LIN {X -0.073,Y -233.852,Z 1712.235,A 0.000,B 0.000,C 90.000,E1 42.285} C_DIS
LIN {X -0.119,Y -224.509,Z 1712.218,A 0.000,B 0.000,C 90.000,E1 39.277} C_DIS
LIN {X 0.012,Y -216.138,Z 1712.201,A 0.000,B 0.000,C 90.000,E1 36.171} C_DIS
LIN {X 0.036,Y -208.461,Z 1712.184,A 0.000,B 0.000,C 90.000,E1 33.038} C_DIS
LIN {X -0.006,Y -201.606,Z 1712.166,A 0.000,B 0.000,C 90.000,E1 29.873} C_DIS
LIN {X 0.104,Y -195.298,Z 1712.148,A 0.000,B 0.000,C 90.000,E1 26.616} C_DIS
LIN {X -0.043,Y -188.244,Z 1712.125,A 0.000,B 0.000,C 90.000,E1 22.567} C_DIS
LIN {X 0.061,Y -183.297,Z 1712.107,A 0.000,B 0.000,C 90.000,E1 19.214} C_DIS
LIN {X -0.070,Y -179.154,Z 1712.088,A 0.000,B 0.000,C 90.000,E1 15.898} C_DIS
LIN {X -0.070,Y -174.908,Z 1712.065,A 0.000,B 0.000,C 90.000,E1 11.658} C_DIS
LIN {X 0.007,Y -171.641,Z 1712.041,A 0.000,B 0.000,C 90.000,E1 7.352} C_DIS
LIN {X -0.001,Y -169.062,Z 1712.012,A 0.000,B 0.000,C 90.000,E1 2.178} C_DIS
LIN {X 0.004,Y -167.943,Z 1711.964,A 0.000,B 0.000,C 90.000,E1 353.451} C_DIS
LIN {X -0.010,Y -169.850,Z 1711.920,A 0.000,B 0.000,C 90.000,E1 345.644} C_DIS
LIN {X -0.055,Y -172.730,Z 1711.891,A 0.000,B 0.000,C 90.000,E1 340.477} C_DIS
LIN {X -0.022,Y -176.262,Z 1711.868,A 0.000,B 0.000,C 90.000,E1 336.177} C_DIS
LIN {X 0.067,Y -180.723,Z 1711.844,A 0.000,B 0.000,C 90.000,E1 331.897} C_DIS
LIN {X 0.046,Y -185.271,Z 1711.825,A 0.000,B 0.000,C 90.000,E1 328.535} C_DIS
LIN {X -0.042,Y -190.788,Z 1711.807,A 0.000,B 0.000,C 90.000,E1 325.229} C_DIS
LIN {X -0.067,Y -195.689,Z 1711.793,A 0.000,B 0.000,C 90.000,E1 322.763} C_DIS
LIN {X -0.052,Y -202.307,Z 1711.777,A 0.000,B 0.000,C 90.000,E1 319.908} C_DIS
LIN {X 0.059,Y -208.732,Z 1711.764,A 0.000,B 0.000,C 90.000,E1 317.472} C_DIS
LIN {X -0.120,Y -217.156,Z 1711.748,A 0.000,B 0.000,C 90.000,E1 314.757} C_DIS
LIN {X -0.028,Y -225.299,Z 1711.736,A 0.000,B 0.000,C 90.000,E1 312.405} C_DIS
LIN {X 0.075,Y -234.395,Z 1711.723,A 0.000,B 0.000,C 90.000,E1 310.092} C_DIS
LIN {X -0.084,Y -242.909,Z 1711.712,A 0.000,B 0.000,C 90.000,E1 308.257} C_DIS
LIN {X 0.079,Y -250.460,Z 1711.704,A 0.000,B 0.000,C 90.000,E1 306.744} C_DIS
LIN {X -0.098,Y -262.879,Z 1711.692,A 0.000,B 0.000,C 90.000,E1 304.612} C_DIS
LIN {X -0.104,Y -281.105,Z 1711.677,A 0.000,B 0.000,C 90.000,E1 301.799} C_DIS
LIN {X -0.081,Y -300.693,Z 1711.661,A 0.000,B 0.000,C 90.000,E1 299.077} C_DIS
LIN {X 0.056,Y -315.955,Z 1711.651,A 0.000,B 0.000,C 90.000,E1 297.078} C_DIS
LIN {X 0.065,Y -331.490,Z 1711.640,A 0.000,B 0.000,C 90.000,E1 295.155} C_DIS
LIN {X 0.085,Y -344.408,Z 1711.631,A 0.000,B 0.000,C 90.000,E1 293.590} C_DIS
LIN {X 0.027,Y -359.701,Z 1711.621,A 0.000,B 0.000,C 90.000,E1 291.770} C_DIS
LIN {X -0.109,Y -371.942,Z 1711.613,A 0.000,B 0.000,C 90.000,E1 290.301} C_DIS
LIN {X 0.053,Y -378.776,Z 1711.608,A 0.000,B 0.000,C 90.000,E1 289.396} C_DIS
LIN {X -0.069,Y -384.788,Z 1711.603,A 0.000,B 0.000,C 90.000,E1 288.544} C_DIS
LIN {X 0.083,Y -388.314,Z 1711.600,A 0.000,B 0.000,C 90.000,E1 287.946} C_DIS
LIN {X -0.112,Y -391.399,Z 1711.597,A 0.000,B 0.000,C 90.000,E1 287.402} C_DIS
LIN {X 0.087,Y -394.052,Z 1711.593,A 0.000,B 0.000,C 90.000,E1 286.804} C_DIS
LIN {X -0.017,Y -397.255,Z 1711.589,A 0.000,B 0.000,C 90.000,E1 285.969} C_DIS
LIN {X -0.162,Y -398.955,Z 1711.586,A 0.000,B 0.000,C 90.000,E1 285.426} C_DIS
LIN {X 0.082,Y -400.312,Z 1711.582,A 0.000,B 0.000,C 90.000,E1 284.828} C_DIS
LIN {X -0.154,Y -401.245,Z 1711.579,A 0.000,B 0.000,C 90.000,E1 284.300} C_DIS
LIN {X 0.011,Y -401.838,Z 1711.576,A 0.000,B 0.000,C 90.000,E1 283.716} C_DIS
LIN {X -0.115,Y -402.031,Z 1711.573,A 0.000,B 0.000,C 90.000,E1 283.175} C_DIS
LIN {X 0.060,Y -401.772,Z 1711.570,A 0.000,B 0.000,C 90.000,E1 282.591} C_DIS
LIN {X -0.154,Y -401.091,Z 1711.567,A 0.000,B 0.000,C 90.000,E1 282.063} C_DIS
LIN {X 0.023,Y -399.884,Z 1711.564,A 0.000,B 0.000,C 90.000,E1 281.478} C_DIS
LIN {X 0.194,Y -398.188,Z 1711.561,A 0.000,B 0.000,C 90.000,E1 280.894} C_DIS
LIN {X -0.034,Y -395.932,Z 1711.558,A 0.000,B 0.000,C 90.000,E1 280.366} C_DIS
LIN {X 0.044,Y -393.111,Z 1711.554,A 0.000,B 0.000,C 90.000,E1 279.792} C_DIS
LIN {X -0.158,Y -388.091,Z 1711.550,A 0.000,B 0.000,C 90.000,E1 278.973} C_DIS
LIN {X -0.066,Y -379.299,Z 1711.542,A 0.000,B 0.000,C 90.000,E1 277.530} C_DIS
LIN {X -0.066,Y -373.299,Z 1711.537,A 0.000,B 0.000,C 90.000,E1 276.663} C_DIS
LIN {X -0.107,Y -368.624,Z 1711.534,A 0.000,B 0.000,C 90.000,E1 276.087} C_DIS
LIN {X -0.152,Y -363.231,Z 1711.531,A 0.000,B 0.000,C 90.000,E1 275.511} C_DIS
LIN {X -0.040,Y -357.396,Z 1711.527,A 0.000,B 0.000,C 90.000,E1 274.935} C_DIS
LIN {X -0.006,Y -351.283,Z 1711.525,A 0.000,B 0.000,C 90.000,E1 274.416} C_DIS
LIN {X -0.054,Y -345.014,Z 1711.522,A 0.000,B 0.000,C 90.000,E1 273.955} C_DIS
LIN {X 0.142,Y -338.578,Z 1711.520,A 0.000,B 0.000,C 90.000,E1 273.498} C_DIS
LIN {X -0.083,Y -332.051,Z 1711.517,A 0.000,B 0.000,C 90.000,E1 273.154} C_DIS
LIN {X -0.060,Y -325.544,Z 1711.516,A 0.000,B 0.000,C 90.000,E1 272.808} C_DIS
LIN {X 0.149,Y -318.882,Z 1711.514,A 0.000,B 0.000,C 90.000,E1 272.465} C_DIS
LIN {X -0.098,Y -312.037,Z 1711.512,A 0.000,B 0.000,C 90.000,E1 272.236} C_DIS
LIN {X -0.141,Y -301.639,Z 1711.510,A 0.000,B 0.000,C 90.000,E1 271.892} C_DIS
LIN {X 0.131,Y -290.878,Z 1711.509,A 0.000,B 0.000,C 90.000,E1 271.547} C_DIS
LIN {X 0.080,Y -279.215,Z 1711.507,A 0.000,B 0.000,C 90.000,E1 271.318} C_DIS
LIN {X -0.015,Y -266.610,Z 1711.506,A 0.000,B 0.000,C 90.000,E1 271.146} C_DIS
LIN {X 0.035,Y -256.490,Z 1711.506,A 0.000,B 0.000,C 90.000,E1 271.031} C_DIS
LIN {X 0.100,Y -247.221,Z 1711.505,A 0.000,B 0.000,C 90.000,E1 270.974} C_DIS
LIN {X 0.052,Y -181.458,Z 1711.505,A 0.000,B 0.000,C 90.000,E1 270.974} C_DIS
LIN {X -0.077,Y -181.557,Z 1711.500,A 0.000,B 0.000,C 90.000,E1 270.000} C_DIS
LIN {X -0.075,Y -180.789,Z 1711.471,A 0.000,B 0.000,C 90.000,E1 264.780} C_DIS
LIN {X 0.000,Y -178.887,Z 1711.443,A 0.000,B 0.000,C 90.000,E1 259.690} C_DIS
LIN {X 0.075,Y -175.930,Z 1711.414,A 0.000,B 0.000,C 90.000,E1 254.574} C_DIS
LIN {X 0.020,Y -175.373,Z 1711.410,A 0.000,B 0.000,C 90.000,E1 253.740} C_DIS
LIN {X 0.079,Y -172.149,Z 1711.386,A 0.000,B 0.000,C 90.000,E1 249.444} C_DIS
LIN {X 0.056,Y -171.615,Z 1711.381,A 0.000,B 0.000,C 90.000,E1 248.592} C_DIS
LIN {X 0.044,Y -167.837,Z 1711.357,A 0.000,B 0.000,C 90.000,E1 244.280} C_DIS
LIN {X 0.061,Y -166.564,Z 1711.348,A 0.000,B 0.000,C 90.000,E1 242.538} C_DIS
LIN {X -0.029,Y -162.558,Z 1711.323,A 0.000,B 0.000,C 90.000,E1 238.201} C_DIS
LIN {X 0.031,Y -161.237,Z 1711.313,A 0.000,B 0.000,C 90.000,E1 236.421} C_DIS
LIN {X 0.065,Y -157.242,Z 1711.289,A 0.000,B 0.000,C 90.000,E1 231.984} C_DIS
LIN {X -0.012,Y -155.965,Z 1711.279,A 0.000,B 0.000,C 90.000,E1 230.231} C_DIS
LIN {X 0.046,Y -152.220,Z 1711.254,A 0.000,B 0.000,C 90.000,E1 225.729} C_DIS
LIN {X 0.067,Y -150.463,Z 1711.239,A 0.000,B 0.000,C 90.000,E1 223.014} C_DIS
LIN {X -0.022,Y -147.188,Z 1711.214,A 0.000,B 0.000,C 90.000,E1 218.508} C_DIS
LIN {X 0.059,Y -145.207,Z 1711.194,A 0.000,B 0.000,C 90.000,E1 214.818} C_DIS
LIN {X -0.031,Y -142.341,Z 1711.163,A 0.000,B 0.000,C 90.000,E1 209.333} C_DIS
LIN {X 0.022,Y -141.730,Z 1711.153,A 0.000,B 0.000,C 90.000,E1 207.462} C_DIS
LIN {X 0.004,Y -139.482,Z 1711.117,A 0.000,B 0.000,C 90.000,E1 200.972} C_DIS
LIN {X -0.007,Y -138.982,Z 1711.101,A 0.000,B 0.000,C 90.000,E1 198.181} C_DIS
LIN {X -0.045,Y -138.333,Z 1711.054,A 0.000,B 0.000,C 90.000,E1 189.792} C_DIS
LIN {X -0.022,Y -139.428,Z 1711.008,A 0.000,B 0.000,C 90.000,E1 181.375} C_DIS
LIN {X 0.032,Y -141.353,Z 1710.971,A 0.000,B 0.000,C 90.000,E1 174.837} C_DIS
LIN {X 0.008,Y -142.706,Z 1710.956,A 0.000,B 0.000,C 90.000,E1 172.064} C_DIS
LIN {X -0.033,Y -145.079,Z 1710.930,A 0.000,B 0.000,C 90.000,E1 167.465} C_DIS
LIN {X -0.038,Y -147.704,Z 1710.910,A 0.000,B 0.000,C 90.000,E1 163.795} C_DIS
LIN {X 0.047,Y -150.357,Z 1710.890,A 0.000,B 0.000,C 90.000,E1 160.115} C_DIS
LIN {X 0.066,Y -153.782,Z 1710.870,A 0.000,B 0.000,C 90.000,E1 156.485} C_DIS
LIN {X -0.015,Y -157.194,Z 1710.849,A 0.000,B 0.000,C 90.000,E1 152.922} C_DIS
LIN {X 0.068,Y -161.354,Z 1710.830,A 0.000,B 0.000,C 90.000,E1 149.331} C_DIS
LIN {X 0.079,Y -165.557,Z 1710.810,A 0.000,B 0.000,C 90.000,E1 145.801} C_DIS
LIN {X -0.037,Y -170.473,Z 1710.791,A 0.000,B 0.000,C 90.000,E1 142.351} C_DIS
LIN {X 0.113,Y -175.355,Z 1710.772,A 0.000,B 0.000,C 90.000,E1 138.852} C_DIS
LIN {X -0.024,Y -180.979,Z 1710.753,A 0.000,B 0.000,C 90.000,E1 135.486} C_DIS
LIN {X -0.037,Y -186.404,Z 1710.734,A 0.000,B 0.000,C 90.000,E1 132.123} C_DIS
LIN {X -0.098,Y -191.032,Z 1710.720,A 0.000,B 0.000,C 90.000,E1 129.644} C_DIS
LIN {X 0.094,Y -196.814,Z 1710.702,A 0.000,B 0.000,C 90.000,E1 126.297} C_DIS
LIN {X 0.013,Y -200.068,Z 1710.693,A 0.000,B 0.000,C 90.000,E1 124.692} C_DIS
LIN {X 0.007,Y -207.567,Z 1710.670,A 0.000,B 0.000,C 90.000,E1 120.669} C_DIS
LIN {X -0.063,Y -209.260,Z 1710.666,A 0.000,B 0.000,C 90.000,E1 119.873} C_DIS
LIN {X -0.135,Y -332.673,Z 1710.666,A 0.000,B 0.000,C 90.000,E1 119.873} C_DIS
LIN {X 0.115,Y -334.980,Z 1710.666,A 0.000,B 0.000,C 90.000,E1 119.795} C_DIS
LIN {X 0.082,Y -339.177,Z 1710.665,A 0.000,B 0.000,C 90.000,E1 119.617} C_DIS
LIN {X -0.082,Y -341.592,Z 1710.664,A 0.000,B 0.000,C 90.000,E1 119.461} C_DIS
LIN {X 0.017,Y -344.886,Z 1710.661,A 0.000,B 0.000,C 90.000,E1 119.077} C_DIS
LIN {X 0.075,Y -346.788,Z 1710.660,A 0.000,B 0.000,C 90.000,E1 118.771} C_DIS
LIN {X -0.129,Y -350.995,Z 1710.655,A 0.000,B 0.000,C 90.000,E1 117.897} C_DIS
LIN {X 0.064,Y -364.150,Z 1710.640,A 0.000,B 0.000,C 90.000,E1 115.155} C_DIS
LIN {X -0.005,Y -378.851,Z 1710.625,A 0.000,B 0.000,C 90.000,E1 112.514} C_DIS
LIN {X 0.106,Y -393.315,Z 1710.612,A 0.000,B 0.000,C 90.000,E1 110.194} C_DIS
LIN {X 0.084,Y -409.198,Z 1710.600,A 0.000,B 0.000,C 90.000,E1 107.946} C_DIS
LIN {X -0.207,Y -426.609,Z 1710.588,A 0.000,B 0.000,C 90.000,E1 105.788} C_DIS
LIN {X -0.198,Y -445.654,Z 1710.576,A 0.000,B 0.000,C 90.000,E1 103.647} C_DIS
LIN {X 0.226,Y -465.672,Z 1710.565,A 0.000,B 0.000,C 90.000,E1 101.591} C_DIS
LIN {X 0.014,Y -488.822,Z 1710.553,A 0.000,B 0.000,C 90.000,E1 99.557} C_DIS
LIN {X 0.092,Y -504.598,Z 1710.546,A 0.000,B 0.000,C 90.000,E1 98.276} C_DIS
LIN {X -0.221,Y -507.002,Z 1710.545,A 0.000,B 0.000,C 90.000,E1 98.106} C_DIS
LIN {X 0.003,Y -510.391,Z 1710.542,A 0.000,B 0.000,C 90.000,E1 97.644} C_DIS
LIN {X -0.052,Y -511.618,Z 1710.541,A 0.000,B 0.000,C 90.000,E1 97.409} C_DIS
LIN {X -0.173,Y -512.507,Z 1710.540,A 0.000,B 0.000,C 90.000,E1 97.182} C_DIS
LIN {X 0.186,Y -513.424,Z 1710.537,A 0.000,B 0.000,C 90.000,E1 96.663} C_DIS
LIN {X 0.040,Y -513.316,Z 1710.534,A 0.000,B 0.000,C 90.000,E1 96.201} C_DIS
LIN {X -0.102,Y -512.160,Z 1710.532,A 0.000,B 0.000,C 90.000,E1 95.739} C_DIS
LIN {X -0.197,Y -511.132,Z 1710.531,A 0.000,B 0.000,C 90.000,E1 95.511} C_DIS
LIN {X -0.244,Y -509.734,Z 1710.529,A 0.000,B 0.000,C 90.000,E1 95.277} C_DIS
LIN {X 0.075,Y -497.149,Z 1710.520,A 0.000,B 0.000,C 90.000,E1 93.555} C_DIS
LIN {X 0.125,Y -484.524,Z 1710.510,A 0.000,B 0.000,C 90.000,E1 91.835} C_DIS
LIN {X -0.077,Y -471.809,Z 1710.501,A 0.000,B 0.000,C 90.000,E1 90.115} C_DIS
LIN {X -0.063,Y -458.968,Z 1710.491,A 0.000,B 0.000,C 90.000,E1 88.339} C_DIS
LIN {X 0.168,Y -445.987,Z 1710.481,A 0.000,B 0.000,C 90.000,E1 86.502} C_DIS
LIN {X 0.139,Y -433.000,Z 1710.470,A 0.000,B 0.000,C 90.000,E1 84.666} C_DIS
LIN {X 0.168,Y -416.433,Z 1710.457,A 0.000,B 0.000,C 90.000,E1 82.243} C_DIS
LIN {X 0.081,Y -397.068,Z 1710.440,A 0.000,B 0.000,C 90.000,E1 79.218} C_DIS
LIN {X -0.139,Y -382.139,Z 1710.426,A 0.000,B 0.000,C 90.000,E1 76.700} C_DIS
LIN {X -0.205,Y -367.739,Z 1710.411,A 0.000,B 0.000,C 90.000,E1 74.102} C_DIS
LIN {X 0.047,Y -355.320,Z 1710.398,A 0.000,B 0.000,C 90.000,E1 71.692} C_DIS
LIN {X 0.136,Y -340.409,Z 1710.381,A 0.000,B 0.000,C 90.000,E1 68.646} C_DIS
LIN {X 0.072,Y -328.886,Z 1710.368,A 0.000,B 0.000,C 90.000,E1 66.177} C_DIS
LIN {X 0.050,Y -316.355,Z 1710.352,A 0.000,B 0.000,C 90.000,E1 63.332} C_DIS
LIN {X -0.197,Y -305.422,Z 1710.338,A 0.000,B 0.000,C 90.000,E1 60.795} C_DIS
LIN {X 0.010,Y -294.627,Z 1710.323,A 0.000,B 0.000,C 90.000,E1 58.122} C_DIS
LIN {X 0.135,Y -286.448,Z 1710.312,A 0.000,B 0.000,C 90.000,E1 56.087} C_DIS
LIN {X 0.022,Y -278.092,Z 1710.300,A 0.000,B 0.000,C 90.000,E1 54.069} C_DIS
LIN {X -0.041,Y -268.222,Z 1710.287,A 0.000,B 0.000,C 90.000,E1 51.662} C_DIS
LIN {X 0.050,Y -258.392,Z 1710.273,A 0.000,B 0.000,C 90.000,E1 49.175} C_DIS
LIN {X 0.053,Y -247.517,Z 1710.257,A 0.000,B 0.000,C 90.000,E1 46.296} C_DIS
LIN {X -0.064,Y -235.971,Z 1710.239,A 0.000,B 0.000,C 90.000,E1 43.014} C_DIS
LIN {X -0.134,Y -225.354,Z 1710.220,A 0.000,B 0.000,C 90.000,E1 39.644} C_DIS
LIN {X -0.060,Y -215.903,Z 1710.201,A 0.000,B 0.000,C 90.000,E1 36.171} C_DIS
LIN {X -0.039,Y -208.266,Z 1710.183,A 0.000,B 0.000,C 90.000,E1 33.038} C_DIS
LIN {X -0.082,Y -201.421,Z 1710.166,A 0.000,B 0.000,C 90.000,E1 29.873} C_DIS
LIN {X 0.026,Y -195.152,Z 1710.148,A 0.000,B 0.000,C 90.000,E1 26.616} C_DIS
LIN {X 0.051,Y -188.122,Z 1710.125,A 0.000,B 0.000,C 90.000,E1 22.514} C_DIS
LIN {X -0.020,Y -183.190,Z 1710.107,A 0.000,B 0.000,C 90.000,E1 19.214} C_DIS
LIN {X 0.021,Y -179.067,Z 1710.088,A 0.000,B 0.000,C 90.000,E1 15.843} C_DIS
LIN {X 0.055,Y -174.829,Z 1710.064,A 0.000,B 0.000,C 90.000,E1 11.591} C_DIS
LIN {X -0.076,Y -171.580,Z 1710.041,A 0.000,B 0.000,C 90.000,E1 7.352} C_DIS
LIN {X -0.085,Y -169.011,Z 1710.012,A 0.000,B 0.000,C 90.000,E1 2.178} C_DIS
LIN {X 0.002,Y -167.882,Z 1709.964,A 0.000,B 0.000,C 90.000,E1 353.451} C_DIS
LIN {X -0.017,Y -169.793,Z 1709.920,A 0.000,B 0.000,C 90.000,E1 345.644} C_DIS
LIN {X 0.099,Y -172.653,Z 1709.891,A 0.000,B 0.000,C 90.000,E1 340.423} C_DIS
LIN {X -0.032,Y -176.218,Z 1709.868,A 0.000,B 0.000,C 90.000,E1 336.177} C_DIS
LIN {X 0.055,Y -180.714,Z 1709.844,A 0.000,B 0.000,C 90.000,E1 331.897} C_DIS
LIN {X 0.033,Y -185.287,Z 1709.825,A 0.000,B 0.000,C 90.000,E1 328.535} C_DIS
LIN {X 0.102,Y -190.854,Z 1709.807,A 0.000,B 0.000,C 90.000,E1 325.182} C_DIS
LIN {X -0.079,Y -195.788,Z 1709.793,A 0.000,B 0.000,C 90.000,E1 322.763} C_DIS
LIN {X -0.062,Y -202.412,Z 1709.777,A 0.000,B 0.000,C 90.000,E1 319.908} C_DIS
LIN {X 0.050,Y -208.879,Z 1709.764,A 0.000,B 0.000,C 90.000,E1 317.472} C_DIS
LIN {X 0.027,Y -217.335,Z 1709.748,A 0.000,B 0.000,C 90.000,E1 314.717} C_DIS
LIN {X -0.031,Y -225.515,Z 1709.736,A 0.000,B 0.000,C 90.000,E1 312.405} C_DIS
LIN {X 0.077,Y -234.626,Z 1709.723,A 0.000,B 0.000,C 90.000,E1 310.092} C_DIS
LIN {X -0.078,Y -243.148,Z 1709.712,A 0.000,B 0.000,C 90.000,E1 308.257} C_DIS
LIN {X -0.113,Y -250.680,Z 1709.704,A 0.000,B 0.000,C 90.000,E1 306.790} C_DIS
LIN {X -0.084,Y -263.090,Z 1709.692,A 0.000,B 0.000,C 90.000,E1 304.612} C_DIS
LIN {X -0.085,Y -281.271,Z 1709.677,A 0.000,B 0.000,C 90.000,E1 301.799} C_DIS
LIN {X -0.055,Y -300.825,Z 1709.661,A 0.000,B 0.000,C 90.000,E1 299.077} C_DIS
LIN {X 0.085,Y -316.083,Z 1709.651,A 0.000,B 0.000,C 90.000,E1 297.078} C_DIS
LIN {X 0.099,Y -331.545,Z 1709.640,A 0.000,B 0.000,C 90.000,E1 295.155} C_DIS
LIN {X -0.196,Y -344.452,Z 1709.631,A 0.000,B 0.000,C 90.000,E1 293.643} C_DIS
LIN {X 0.100,Y -359.701,Z 1709.621,A 0.000,B 0.000,C 90.000,E1 291.770} C_DIS
LIN {X -0.123,Y -369.594,Z 1709.614,A 0.000,B 0.000,C 90.000,E1 290.610} C_DIS
LIN {X 0.023,Y -376.566,Z 1709.609,A 0.000,B 0.000,C 90.000,E1 289.704} C_DIS
LIN {X -0.116,Y -380.869,Z 1709.606,A 0.000,B 0.000,C 90.000,E1 289.141} C_DIS
LIN {X 0.007,Y -384.821,Z 1709.603,A 0.000,B 0.000,C 90.000,E1 288.544} C_DIS
LIN {X -0.211,Y -388.386,Z 1709.600,A 0.000,B 0.000,C 90.000,E1 288.000} C_DIS
LIN {X -0.035,Y -391.476,Z 1709.597,A 0.000,B 0.000,C 90.000,E1 287.402} C_DIS
LIN {X 0.164,Y -394.104,Z 1709.594,A 0.000,B 0.000,C 90.000,E1 286.804} C_DIS
LIN {X 0.060,Y -397.394,Z 1709.589,A 0.000,B 0.000,C 90.000,E1 285.969} C_DIS
LIN {X -0.082,Y -399.087,Z 1709.586,A 0.000,B 0.000,C 90.000,E1 285.426} C_DIS
LIN {X 0.163,Y -400.457,Z 1709.583,A 0.000,B 0.000,C 90.000,E1 284.828} C_DIS
LIN {X -0.072,Y -401.431,Z 1709.579,A 0.000,B 0.000,C 90.000,E1 284.300} C_DIS
LIN {X 0.094,Y -402.004,Z 1709.576,A 0.000,B 0.000,C 90.000,E1 283.716} C_DIS
LIN {X -0.031,Y -402.214,Z 1709.573,A 0.000,B 0.000,C 90.000,E1 283.175} C_DIS
LIN {X 0.145,Y -401.980,Z 1709.570,A 0.000,B 0.000,C 90.000,E1 282.591} C_DIS
LIN {X -0.068,Y -401.298,Z 1709.567,A 0.000,B 0.000,C 90.000,E1 282.063} C_DIS
LIN {X 0.110,Y -400.154,Z 1709.564,A 0.000,B 0.000,C 90.000,E1 281.478} C_DIS
LIN {X -0.109,Y -398.447,Z 1709.561,A 0.000,B 0.000,C 90.000,E1 280.950} C_DIS
LIN {X 0.055,Y -396.218,Z 1709.558,A 0.000,B 0.000,C 90.000,E1 280.366} C_DIS
LIN {X 0.134,Y -393.406,Z 1709.555,A 0.000,B 0.000,C 90.000,E1 279.792} C_DIS
LIN {X -0.066,Y -388.456,Z 1709.550,A 0.000,B 0.000,C 90.000,E1 278.973} C_DIS
LIN {X 0.029,Y -379.616,Z 1709.542,A 0.000,B 0.000,C 90.000,E1 277.530} C_DIS
LIN {X 0.030,Y -373.544,Z 1709.537,A 0.000,B 0.000,C 90.000,E1 276.663} C_DIS
LIN {X -0.011,Y -368.837,Z 1709.534,A 0.000,B 0.000,C 90.000,E1 276.087} C_DIS
LIN {X -0.062,Y -363.443,Z 1709.531,A 0.000,B 0.000,C 90.000,E1 275.511} C_DIS
LIN {X 0.058,Y -357.562,Z 1709.527,A 0.000,B 0.000,C 90.000,E1 274.935} C_DIS
LIN {X 0.116,Y -351.452,Z 1709.525,A 0.000,B 0.000,C 90.000,E1 274.416} C_DIS
LIN {X 0.084,Y -345.215,Z 1709.522,A 0.000,B 0.000,C 90.000,E1 273.955} C_DIS
LIN {X -0.049,Y -338.811,Z 1709.520,A 0.000,B 0.000,C 90.000,E1 273.555} C_DIS
LIN {X 0.075,Y -332.277,Z 1709.518,A 0.000,B 0.000,C 90.000,E1 273.154} C_DIS
LIN {X 0.096,Y -325.680,Z 1709.516,A 0.000,B 0.000,C 90.000,E1 272.808} C_DIS
LIN {X -0.034,Y -318.935,Z 1709.514,A 0.000,B 0.000,C 90.000,E1 272.522} C_DIS
LIN {X 0.041,Y -312.097,Z 1709.512,A 0.000,B 0.000,C 90.000,E1 272.236} C_DIS
LIN {X 0.020,Y -301.843,Z 1709.510,A 0.000,B 0.000,C 90.000,E1 271.892} C_DIS
LIN {X -0.010,Y -291.070,Z 1709.509,A 0.000,B 0.000,C 90.000,E1 271.604} C_DIS
LIN {X -0.052,Y -279.680,Z 1709.508,A 0.000,B 0.000,C 90.000,E1 271.375} C_DIS
LIN {X 0.113,Y -267.186,Z 1709.506,A 0.000,B 0.000,C 90.000,E1 271.146} C_DIS
LIN {X -0.102,Y -256.616,Z 1709.506,A 0.000,B 0.000,C 90.000,E1 271.088} C_DIS
LIN {X -0.031,Y -247.213,Z 1709.506,A 0.000,B 0.000,C 90.000,E1 271.031} C_DIS
LIN {X -0.045,Y -181.452,Z 1709.506,A 0.000,B 0.000,C 90.000,E1 271.031} C_DIS
LIN {X 0.008,Y -181.561,Z 1709.500,A 0.000,B 0.000,C 90.000,E1 270.000} C_DIS
LIN {X 0.010,Y -180.799,Z 1709.471,A 0.000,B 0.000,C 90.000,E1 264.780} C_DIS
LIN {X 0.083,Y -178.899,Z 1709.443,A 0.000,B 0.000,C 90.000,E1 259.690} C_DIS
LIN {X -0.012,Y -175.941,Z 1709.415,A 0.000,B 0.000,C 90.000,E1 254.629} C_DIS
LIN {X -0.065,Y -175.398,Z 1709.410,A 0.000,B 0.000,C 90.000,E1 253.795} C_DIS
LIN {X -0.061,Y -172.166,Z 1709.386,A 0.000,B 0.000,C 90.000,E1 249.518} C_DIS
LIN {X -0.022,Y -171.635,Z 1709.381,A 0.000,B 0.000,C 90.000,E1 248.646} C_DIS
LIN {X -0.026,Y -167.858,Z 1709.357,A 0.000,B 0.000,C 90.000,E1 244.332} C_DIS
LIN {X -0.083,Y -166.590,Z 1709.348,A 0.000,B 0.000,C 90.000,E1 242.615} C_DIS
LIN {X 0.051,Y -162.580,Z 1709.323,A 0.000,B 0.000,C 90.000,E1 238.201} C_DIS
LIN {X 0.020,Y -161.262,Z 1709.314,A 0.000,B 0.000,C 90.000,E1 236.453} C_DIS
LIN {X 0.019,Y -157.263,Z 1709.289,A 0.000,B 0.000,C 90.000,E1 232.029} C_DIS
LIN {X -0.055,Y -155.984,Z 1709.279,A 0.000,B 0.000,C 90.000,E1 230.275} C_DIS
LIN {X -0.093,Y -152.241,Z 1709.254,A 0.000,B 0.000,C 90.000,E1 225.810} C_DIS
LIN {X 0.033,Y -150.481,Z 1709.239,A 0.000,B 0.000,C 90.000,E1 223.056} C_DIS
LIN {X -0.040,Y -147.206,Z 1709.214,A 0.000,B 0.000,C 90.000,E1 218.543} C_DIS
LIN {X -0.069,Y -145.226,Z 1709.194,A 0.000,B 0.000,C 90.000,E1 214.898} C_DIS
LIN {X 0.041,Y -142.352,Z 1709.163,A 0.000,B 0.000,C 90.000,E1 209.333} C_DIS
LIN {X -0.031,Y -141.740,Z 1709.153,A 0.000,B 0.000,C 90.000,E1 207.513} C_DIS
LIN {X 0.076,Y -139.487,Z 1709.117,A 0.000,B 0.000,C 90.000,E1 200.972} C_DIS
LIN {X 0.064,Y -138.989,Z 1709.101,A 0.000,B 0.000,C 90.000,E1 198.181} C_DIS
LIN {X 0.026,Y -138.335,Z 1709.054,A 0.000,B 0.000,C 90.000,E1 189.792} C_DIS
LIN {X 0.050,Y -139.420,Z 1709.008,A 0.000,B 0.000,C 90.000,E1 181.375} C_DIS
LIN {X -0.037,Y -141.339,Z 1708.972,A 0.000,B 0.000,C 90.000,E1 174.894} C_DIS
LIN {X -0.079,Y -142.695,Z 1708.956,A 0.000,B 0.000,C 90.000,E1 172.129} C_DIS
LIN {X 0.041,Y -145.061,Z 1708.930,A 0.000,B 0.000,C 90.000,E1 167.465} C_DIS
LIN {X 0.038,Y -147.686,Z 1708.910,A 0.000,B 0.000,C 90.000,E1 163.795} C_DIS
LIN {X -0.070,Y -150.334,Z 1708.890,A 0.000,B 0.000,C 90.000,E1 160.188} C_DIS
LIN {X 0.001,Y -153.751,Z 1708.870,A 0.000,B 0.000,C 90.000,E1 156.538} C_DIS
LIN {X -0.008,Y -157.164,Z 1708.850,A 0.000,B 0.000,C 90.000,E1 152.948} C_DIS
LIN {X -0.074,Y -161.318,Z 1708.830,A 0.000,B 0.000,C 90.000,E1 149.410} C_DIS
LIN {X 0.080,Y -164.432,Z 1708.815,A 0.000,B 0.000,C 90.000,E1 146.707} C_DIS
LIN {X 0.073,Y -169.119,Z 1708.796,A 0.000,B 0.000,C 90.000,E1 143.210} C_DIS
LIN {X 0.022,Y -171.672,Z 1708.786,A 0.000,B 0.000,C 90.000,E1 141.492} C_DIS
LIN {X -0.067,Y -176.640,Z 1708.767,A 0.000,B 0.000,C 90.000,E1 138.081} C_DIS
LIN {X 0.061,Y -180.937,Z 1708.753,A 0.000,B 0.000,C 90.000,E1 135.486} C_DIS
LIN {X 0.050,Y -186.357,Z 1708.734,A 0.000,B 0.000,C 90.000,E1 132.123} C_DIS
LIN {X -0.010,Y -190.988,Z 1708.720,A 0.000,B 0.000,C 90.000,E1 129.644} C_DIS
LIN {X -0.092,Y -196.764,Z 1708.702,A 0.000,B 0.000,C 90.000,E1 126.377} C_DIS
LIN {X -0.061,Y -200.013,Z 1708.693,A 0.000,B 0.000,C 90.000,E1 124.739} C_DIS
LIN {X 0.099,Y -207.516,Z 1708.671,A 0.000,B 0.000,C 90.000,E1 120.669} C_DIS
LIN {X 0.074,Y -209.181,Z 1708.666,A 0.000,B 0.000,C 90.000,E1 119.873} C_DIS
LIN {X 0.083,Y -332.295,Z 1708.666,A 0.000,B 0.000,C 90.000,E1 119.873} C_DIS
LIN {X -0.194,Y -335.216,Z 1708.666,A 0.000,B 0.000,C 90.000,E1 119.873} C_DIS
LIN {X -0.063,Y -339.167,Z 1708.665,A 0.000,B 0.000,C 90.000,E1 119.667} C_DIS
LIN {X 0.069,Y -341.531,Z 1708.664,A 0.000,B 0.000,C 90.000,E1 119.461} C_DIS
LIN {X 0.168,Y -344.782,Z 1708.662,A 0.000,B 0.000,C 90.000,E1 119.077} C_DIS
LIN {X -0.093,Y -346.682,Z 1708.660,A 0.000,B 0.000,C 90.000,E1 118.821} C_DIS
LIN {X 0.011,Y -352.269,Z 1708.653,A 0.000,B 0.000,C 90.000,E1 117.590} C_DIS
LIN {X -0.079,Y -365.583,Z 1708.638,A 0.000,B 0.000,C 90.000,E1 114.899} C_DIS
LIN {X -0.112,Y -380.447,Z 1708.624,A 0.000,B 0.000,C 90.000,E1 112.259} C_DIS
LIN {X 0.029,Y -395.071,Z 1708.611,A 0.000,B 0.000,C 90.000,E1 109.939} C_DIS
LIN {X 0.039,Y -411.126,Z 1708.598,A 0.000,B 0.000,C 90.000,E1 107.692} C_DIS
LIN {X 0.194,Y -428.723,Z 1708.586,A 0.000,B 0.000,C 90.000,E1 105.481} C_DIS
LIN {X 0.191,Y -447.928,Z 1708.574,A 0.000,B 0.000,C 90.000,E1 103.355} C_DIS
LIN {X -0.216,Y -468.013,Z 1708.563,A 0.000,B 0.000,C 90.000,E1 101.422} C_DIS
LIN {X -0.211,Y -491.255,Z 1708.552,A 0.000,B 0.000,C 90.000,E1 99.378} C_DIS
LIN {X 0.203,Y -504.404,Z 1708.546,A 0.000,B 0.000,C 90.000,E1 98.276} C_DIS
LIN {X -0.111,Y -506.800,Z 1708.545,A 0.000,B 0.000,C 90.000,E1 98.106} C_DIS
LIN {X 0.031,Y -508.717,Z 1708.544,A 0.000,B 0.000,C 90.000,E1 97.871} C_DIS
LIN {X 0.104,Y -510.183,Z 1708.542,A 0.000,B 0.000,C 90.000,E1 97.644} C_DIS
LIN {X 0.054,Y -511.402,Z 1708.541,A 0.000,B 0.000,C 90.000,E1 97.409} C_DIS
LIN {X -0.063,Y -512.284,Z 1708.540,A 0.000,B 0.000,C 90.000,E1 97.182} C_DIS
LIN {X -0.215,Y -513.195,Z 1708.537,A 0.000,B 0.000,C 90.000,E1 96.720} C_DIS
LIN {X 0.148,Y -513.081,Z 1708.535,A 0.000,B 0.000,C 90.000,E1 96.201} C_DIS
LIN {X 0.005,Y -511.920,Z 1708.532,A 0.000,B 0.000,C 90.000,E1 95.739} C_DIS
LIN {X -0.091,Y -510.890,Z 1708.531,A 0.000,B 0.000,C 90.000,E1 95.511} C_DIS
LIN {X -0.139,Y -509.488,Z 1708.529,A 0.000,B 0.000,C 90.000,E1 95.277} C_DIS
LIN {X 0.172,Y -496.899,Z 1708.520,A 0.000,B 0.000,C 90.000,E1 93.555} C_DIS
LIN {X 0.214,Y -484.285,Z 1708.510,A 0.000,B 0.000,C 90.000,E1 91.835} C_DIS
LIN {X 0.007,Y -471.582,Z 1708.501,A 0.000,B 0.000,C 90.000,E1 90.115} C_DIS
LIN {X 0.013,Y -458.748,Z 1708.491,A 0.000,B 0.000,C 90.000,E1 88.339} C_DIS
LIN {X -0.207,Y -445.766,Z 1708.481,A 0.000,B 0.000,C 90.000,E1 86.560} C_DIS
LIN {X 0.202,Y -432.745,Z 1708.470,A 0.000,B 0.000,C 90.000,E1 84.666} C_DIS
LIN {X -0.189,Y -416.155,Z 1708.457,A 0.000,B 0.000,C 90.000,E1 82.299} C_DIS
LIN {X 0.124,Y -396.765,Z 1708.440,A 0.000,B 0.000,C 90.000,E1 79.218} C_DIS
LIN {X -0.106,Y -381.820,Z 1708.426,A 0.000,B 0.000,C 90.000,E1 76.700} C_DIS
LIN {X -0.181,Y -367.393,Z 1708.411,A 0.000,B 0.000,C 90.000,E1 74.102} C_DIS
LIN {X 0.061,Y -354.939,Z 1708.398,A 0.000,B 0.000,C 90.000,E1 71.692} C_DIS
LIN {X 0.139,Y -340.019,Z 1708.381,A 0.000,B 0.000,C 90.000,E1 68.646} C_DIS
LIN {X 0.087,Y -329.937,Z 1708.370,A 0.000,B 0.000,C 90.000,E1 66.485} C_DIS
LIN {X 0.103,Y -317.363,Z 1708.354,A 0.000,B 0.000,C 90.000,E1 63.640} C_DIS
LIN {X 0.153,Y -306.425,Z 1708.339,A 0.000,B 0.000,C 90.000,E1 61.051} C_DIS
LIN {X -0.047,Y -296.966,Z 1708.327,A 0.000,B 0.000,C 90.000,E1 58.791} C_DIS
LIN {X -0.031,Y -288.862,Z 1708.315,A 0.000,B 0.000,C 90.000,E1 56.786} C_DIS
LIN {X -0.095,Y -280.542,Z 1708.304,A 0.000,B 0.000,C 90.000,E1 54.769} C_DIS
LIN {X 0.016,Y -272.100,Z 1708.293,A 0.000,B 0.000,C 90.000,E1 52.683} C_DIS
LIN {X 0.032,Y -262.245,Z 1708.279,A 0.000,B 0.000,C 90.000,E1 50.231} C_DIS
LIN {X -0.022,Y -249.840,Z 1708.261,A 0.000,B 0.000,C 90.000,E1 47.025} C_DIS
LIN {X 0.088,Y -238.126,Z 1708.243,A 0.000,B 0.000,C 90.000,E1 43.704} C_DIS
LIN {X 0.068,Y -227.351,Z 1708.224,A 0.000,B 0.000,C 90.000,E1 40.334} C_DIS
LIN {X -0.021,Y -219.737,Z 1708.209,A 0.000,B 0.000,C 90.000,E1 37.684} C_DIS
LIN {X -0.131,Y -211.754,Z 1708.192,A 0.000,B 0.000,C 90.000,E1 34.612} C_DIS
LIN {X 0.020,Y -204.588,Z 1708.175,A 0.000,B 0.000,C 90.000,E1 31.416} C_DIS
LIN {X -0.044,Y -198.055,Z 1708.157,A 0.000,B 0.000,C 90.000,E1 28.231} C_DIS
LIN {X 0.059,Y -192.107,Z 1708.139,A 0.000,B 0.000,C 90.000,E1 24.951} C_DIS
LIN {X 0.045,Y -186.702,Z 1708.120,A 0.000,B 0.000,C 90.000,E1 21.663} C_DIS
LIN {X -0.057,Y -181.998,Z 1708.102,A 0.000,B 0.000,C 90.000,E1 18.362} C_DIS
LIN {X 0.073,Y -178.053,Z 1708.083,A 0.000,B 0.000,C 90.000,E1 14.954} C_DIS
LIN {X 0.035,Y -174.027,Z 1708.060,A 0.000,B 0.000,C 90.000,E1 10.715} C_DIS
LIN {X 0.022,Y -170.474,Z 1708.031,A 0.000,B 0.000,C 90.000,E1 5.568} C_DIS
LIN {X -0.031,Y -168.276,Z 1707.997,A 0.000,B 0.000,C 90.000,E1 359.542} C_DIS
LIN {X 0.000,Y -168.498,Z 1707.939,A 0.000,B 0.000,C 90.000,E1 349.106} C_DIS
LIN {X 0.027,Y -171.009,Z 1707.906,A 0.000,B 0.000,C 90.000,E1 343.032} C_DIS
LIN {X 0.041,Y -173.869,Z 1707.882,A 0.000,B 0.000,C 90.000,E1 338.720} C_DIS
LIN {X -0.010,Y -177.878,Z 1707.858,A 0.000,B 0.000,C 90.000,E1 334.460} C_DIS
LIN {X 0.044,Y -181.753,Z 1707.839,A 0.000,B 0.000,C 90.000,E1 331.051} C_DIS
LIN {X -0.015,Y -186.589,Z 1707.821,A 0.000,B 0.000,C 90.000,E1 327.709} C_DIS
LIN {X 0.089,Y -190.917,Z 1707.807,A 0.000,B 0.000,C 90.000,E1 325.182} C_DIS
LIN {X -0.092,Y -195.884,Z 1707.793,A 0.000,B 0.000,C 90.000,E1 322.763} C_DIS
LIN {X -0.073,Y -202.532,Z 1707.777,A 0.000,B 0.000,C 90.000,E1 319.908} C_DIS
LIN {X 0.041,Y -209.023,Z 1707.764,A 0.000,B 0.000,C 90.000,E1 317.472} C_DIS
LIN {X 0.022,Y -217.521,Z 1707.748,A 0.000,B 0.000,C 90.000,E1 314.717} C_DIS
LIN {X -0.033,Y -225.726,Z 1707.736,A 0.000,B 0.000,C 90.000,E1 312.405} C_DIS
LIN {X 0.127,Y -233.249,Z 1707.725,A 0.000,B 0.000,C 90.000,E1 310.458} C_DIS
LIN {X -0.054,Y -241.616,Z 1707.714,A 0.000,B 0.000,C 90.000,E1 308.624} C_DIS
LIN {X -0.107,Y -248.955,Z 1707.706,A 0.000,B 0.000,C 90.000,E1 307.156} C_DIS
LIN {X 0.039,Y -261.163,Z 1707.694,A 0.000,B 0.000,C 90.000,E1 304.945} C_DIS
LIN {X -0.009,Y -279.108,Z 1707.678,A 0.000,B 0.000,C 90.000,E1 302.133} C_DIS
LIN {X -0.032,Y -298.473,Z 1707.663,A 0.000,B 0.000,C 90.000,E1 299.411} C_DIS
LIN {X -0.070,Y -313.666,Z 1707.652,A 0.000,B 0.000,C 90.000,E1 297.436} C_DIS
LIN {X 0.177,Y -329.021,Z 1707.642,A 0.000,B 0.000,C 90.000,E1 295.463} C_DIS
LIN {X -0.147,Y -341.930,Z 1707.633,A 0.000,B 0.000,C 90.000,E1 293.951} C_DIS
LIN {X 0.099,Y -357.218,Z 1707.623,A 0.000,B 0.000,C 90.000,E1 292.078} C_DIS
LIN {X -0.069,Y -369.627,Z 1707.614,A 0.000,B 0.000,C 90.000,E1 290.610} C_DIS
LIN {X 0.080,Y -376.599,Z 1707.609,A 0.000,B 0.000,C 90.000,E1 289.704} C_DIS
LIN {X -0.058,Y -380.912,Z 1707.606,A 0.000,B 0.000,C 90.000,E1 289.141} C_DIS
LIN {X 0.064,Y -384.854,Z 1707.603,A 0.000,B 0.000,C 90.000,E1 288.544} C_DIS
LIN {X -0.152,Y -388.416,Z 1707.600,A 0.000,B 0.000,C 90.000,E1 288.000} C_DIS
LIN {X 0.177,Y -392.936,Z 1707.595,A 0.000,B 0.000,C 90.000,E1 287.094} C_DIS
LIN {X 0.064,Y -396.505,Z 1707.590,A 0.000,B 0.000,C 90.000,E1 286.260} C_DIS
LIN {X -0.020,Y -399.256,Z 1707.586,A 0.000,B 0.000,C 90.000,E1 285.426} C_DIS
LIN {X 0.226,Y -400.627,Z 1707.583,A 0.000,B 0.000,C 90.000,E1 284.828} C_DIS
LIN {X -0.008,Y -401.628,Z 1707.579,A 0.000,B 0.000,C 90.000,E1 284.300} C_DIS
LIN {X -0.231,Y -402.193,Z 1707.576,A 0.000,B 0.000,C 90.000,E1 283.772} C_DIS
LIN {X 0.036,Y -402.410,Z 1707.573,A 0.000,B 0.000,C 90.000,E1 283.175} C_DIS
LIN {X -0.179,Y -402.187,Z 1707.570,A 0.000,B 0.000,C 90.000,E1 282.647} C_DIS
LIN {X 0.001,Y -401.527,Z 1707.567,A 0.000,B 0.000,C 90.000,E1 282.063} C_DIS
LIN {X 0.179,Y -400.343,Z 1707.564,A 0.000,B 0.000,C 90.000,E1 281.478} C_DIS
LIN {X -0.038,Y -398.717,Z 1707.561,A 0.000,B 0.000,C 90.000,E1 280.950} C_DIS
LIN {X 0.127,Y -396.490,Z 1707.558,A 0.000,B 0.000,C 90.000,E1 280.366} C_DIS
LIN {X -0.182,Y -393.732,Z 1707.555,A 0.000,B 0.000,C 90.000,E1 279.849} C_DIS
LIN {X 0.008,Y -388.813,Z 1707.550,A 0.000,B 0.000,C 90.000,E1 278.973} C_DIS
LIN {X 0.107,Y -379.947,Z 1707.542,A 0.000,B 0.000,C 90.000,E1 277.530} C_DIS
LIN {X 0.110,Y -373.809,Z 1707.537,A 0.000,B 0.000,C 90.000,E1 276.663} C_DIS
LIN {X 0.070,Y -369.019,Z 1707.534,A 0.000,B 0.000,C 90.000,E1 276.087} C_DIS
LIN {X 0.028,Y -363.674,Z 1707.531,A 0.000,B 0.000,C 90.000,E1 275.511} C_DIS
LIN {X -0.182,Y -357.776,Z 1707.528,A 0.000,B 0.000,C 90.000,E1 274.992} C_DIS
LIN {X -0.081,Y -351.693,Z 1707.525,A 0.000,B 0.000,C 90.000,E1 274.473} C_DIS
LIN {X -0.074,Y -345.484,Z 1707.522,A 0.000,B 0.000,C 90.000,E1 274.012} C_DIS
LIN {X 0.136,Y -339.081,Z 1707.520,A 0.000,B 0.000,C 90.000,E1 273.555} C_DIS
LIN {X -0.087,Y -332.487,Z 1707.518,A 0.000,B 0.000,C 90.000,E1 273.212} C_DIS
LIN {X -0.056,Y -325.902,Z 1707.516,A 0.000,B 0.000,C 90.000,E1 272.865} C_DIS
LIN {X 0.148,Y -319.159,Z 1707.514,A 0.000,B 0.000,C 90.000,E1 272.522} C_DIS
LIN {X -0.086,Y -312.380,Z 1707.513,A 0.000,B 0.000,C 90.000,E1 272.293} C_DIS
LIN {X -0.088,Y -302.206,Z 1707.511,A 0.000,B 0.000,C 90.000,E1 271.949} C_DIS
LIN {X -0.113,Y -291.653,Z 1707.509,A 0.000,B 0.000,C 90.000,E1 271.661} C_DIS
LIN {X 0.116,Y -280.363,Z 1707.508,A 0.000,B 0.000,C 90.000,E1 271.375} C_DIS
LIN {X -0.004,Y -268.066,Z 1707.507,A 0.000,B 0.000,C 90.000,E1 271.203} C_DIS
LIN {X 0.039,Y -257.474,Z 1707.506,A 0.000,B 0.000,C 90.000,E1 271.088} C_DIS
LIN {X 0.090,Y -247.909,Z 1707.506,A 0.000,B 0.000,C 90.000,E1 271.031} C_DIS
LIN {X 0.043,Y -181.446,Z 1707.506,A 0.000,B 0.000,C 90.000,E1 271.031} C_DIS
LIN {X -0.089,Y -181.565,Z 1707.500,A 0.000,B 0.000,C 90.000,E1 270.057} C_DIS
LIN {X -0.086,Y -180.808,Z 1707.471,A 0.000,B 0.000,C 90.000,E1 264.837} C_DIS
LIN {X -0.008,Y -178.910,Z 1707.443,A 0.000,B 0.000,C 90.000,E1 259.746} C_DIS
LIN {X 0.071,Y -175.954,Z 1707.415,A 0.000,B 0.000,C 90.000,E1 254.629} C_DIS
LIN {X 0.018,Y -175.422,Z 1707.410,A 0.000,B 0.000,C 90.000,E1 253.795} C_DIS
LIN {X 0.021,Y -172.183,Z 1707.386,A 0.000,B 0.000,C 90.000,E1 249.518} C_DIS
LIN {X 0.061,Y -171.655,Z 1707.381,A 0.000,B 0.000,C 90.000,E1 248.646} C_DIS
LIN {X 0.055,Y -167.879,Z 1707.358,A 0.000,B 0.000,C 90.000,E1 244.332} C_DIS
LIN {X -0.002,Y -166.614,Z 1707.348,A 0.000,B 0.000,C 90.000,E1 242.615} C_DIS
LIN {X -0.008,Y -162.602,Z 1707.324,A 0.000,B 0.000,C 90.000,E1 238.250} C_DIS
LIN {X -0.035,Y -161.287,Z 1707.314,A 0.000,B 0.000,C 90.000,E1 236.501} C_DIS
LIN {X 0.000,Y -157.285,Z 1707.289,A 0.000,B 0.000,C 90.000,E1 232.065} C_DIS
LIN {X 0.023,Y -156.003,Z 1707.279,A 0.000,B 0.000,C 90.000,E1 230.275} C_DIS
LIN {X -0.017,Y -152.261,Z 1707.255,A 0.000,B 0.000,C 90.000,E1 225.810} C_DIS
LIN {X 0.005,Y -150.499,Z 1707.239,A 0.000,B 0.000,C 90.000,E1 223.095} C_DIS
LIN {X 0.035,Y -147.224,Z 1707.214,A 0.000,B 0.000,C 90.000,E1 218.543} C_DIS
LIN {X 0.005,Y -145.246,Z 1707.194,A 0.000,B 0.000,C 90.000,E1 214.898} C_DIS
LIN {X -0.080,Y -142.364,Z 1707.163,A 0.000,B 0.000,C 90.000,E1 209.411} C_DIS
LIN {X 0.042,Y -141.750,Z 1707.153,A 0.000,B 0.000,C 90.000,E1 207.513} C_DIS
LIN {X -0.032,Y -139.494,Z 1707.117,A 0.000,B 0.000,C 90.000,E1 201.046} C_DIS
LIN {X 0.005,Y -138.997,Z 1707.101,A 0.000,B 0.000,C 90.000,E1 198.236} C_DIS
LIN {X -0.039,Y -138.337,Z 1707.055,A 0.000,B 0.000,C 90.000,E1 189.849} C_DIS
LIN {X -0.017,Y -139.413,Z 1707.008,A 0.000,B 0.000,C 90.000,E1 181.432} C_DIS
LIN {X 0.037,Y -141.326,Z 1706.972,A 0.000,B 0.000,C 90.000,E1 174.894} C_DIS
LIN {X -0.006,Y -142.684,Z 1706.956,A 0.000,B 0.000,C 90.000,E1 172.129} C_DIS
LIN {X -0.026,Y -145.042,Z 1706.931,A 0.000,B 0.000,C 90.000,E1 167.521} C_DIS
LIN {X -0.029,Y -147.667,Z 1706.910,A 0.000,B 0.000,C 90.000,E1 163.850} C_DIS
LIN {X 0.006,Y -150.310,Z 1706.890,A 0.000,B 0.000,C 90.000,E1 160.188} C_DIS
LIN {X 0.017,Y -153.721,Z 1706.870,A 0.000,B 0.000,C 90.000,E1 156.561} C_DIS
LIN {X -0.069,Y -157.135,Z 1706.850,A 0.000,B 0.000,C 90.000,E1 152.999} C_DIS
LIN {X 0.005,Y -161.281,Z 1706.830,A 0.000,B 0.000,C 90.000,E1 149.410} C_DIS
LIN {X 0.023,Y -164.399,Z 1706.815,A 0.000,B 0.000,C 90.000,E1 146.755} C_DIS
LIN {X 0.020,Y -169.078,Z 1706.796,A 0.000,B 0.000,C 90.000,E1 143.256} C_DIS
LIN {X -0.029,Y -171.636,Z 1706.786,A 0.000,B 0.000,C 90.000,E1 141.537} C_DIS
LIN {X 0.018,Y -176.596,Z 1706.767,A 0.000,B 0.000,C 90.000,E1 138.081} C_DIS
LIN {X 0.020,Y -180.894,Z 1706.753,A 0.000,B 0.000,C 90.000,E1 135.526} C_DIS
LIN {X 0.011,Y -186.310,Z 1706.734,A 0.000,B 0.000,C 90.000,E1 132.162} C_DIS
LIN {X 0.078,Y -190.944,Z 1706.720,A 0.000,B 0.000,C 90.000,E1 129.644} C_DIS
LIN {X -0.002,Y -196.714,Z 1706.702,A 0.000,B 0.000,C 90.000,E1 126.377} C_DIS
LIN {X 0.029,Y -199.960,Z 1706.693,A 0.000,B 0.000,C 90.000,E1 124.739} C_DIS
LIN {X -0.079,Y -205.875,Z 1706.675,A 0.000,B 0.000,C 90.000,E1 121.544} C_DIS
LIN {X 0.008,Y -209.115,Z 1706.666,A 0.000,B 0.000,C 90.000,E1 119.922} C_DIS
LIN {X -0.023,Y -332.654,Z 1706.666,A 0.000,B 0.000,C 90.000,E1 119.922} C_DIS
LIN {X -0.045,Y -335.366,Z 1706.666,A 0.000,B 0.000,C 90.000,E1 119.873} C_DIS
LIN {X 0.087,Y -339.148,Z 1706.665,A 0.000,B 0.000,C 90.000,E1 119.667} C_DIS
LIN {X 0.052,Y -341.471,Z 1706.664,A 0.000,B 0.000,C 90.000,E1 119.489} C_DIS
LIN {X 0.019,Y -344.681,Z 1706.662,A 0.000,B 0.000,C 90.000,E1 119.127} C_DIS
LIN {X 0.045,Y -346.576,Z 1706.660,A 0.000,B 0.000,C 90.000,E1 118.821} C_DIS
LIN {X 0.002,Y -353.563,Z 1706.652,A 0.000,B 0.000,C 90.000,E1 117.308} C_DIS
LIN {X 0.117,Y -367.028,Z 1706.637,A 0.000,B 0.000,C 90.000,E1 114.591} C_DIS
LIN {X -0.012,Y -382.065,Z 1706.622,A 0.000,B 0.000,C 90.000,E1 111.972} C_DIS
LIN {X -0.049,Y -396.851,Z 1706.609,A 0.000,B 0.000,C 90.000,E1 109.685} C_DIS
LIN {X -0.134,Y -413.080,Z 1706.597,A 0.000,B 0.000,C 90.000,E1 107.457} C_DIS
LIN {X 0.067,Y -430.866,Z 1706.585,A 0.000,B 0.000,C 90.000,E1 105.245} C_DIS
LIN {X 0.142,Y -450.235,Z 1706.573,A 0.000,B 0.000,C 90.000,E1 103.119} C_DIS
LIN {X -0.110,Y -470.387,Z 1706.562,A 0.000,B 0.000,C 90.000,E1 101.186} C_DIS
LIN {X 0.004,Y -493.667,Z 1706.551,A 0.000,B 0.000,C 90.000,E1 99.151} C_DIS
LIN {X -0.257,Y -504.209,Z 1706.546,A 0.000,B 0.000,C 90.000,E1 98.341} C_DIS
LIN {X 0.000,Y -506.596,Z 1706.545,A 0.000,B 0.000,C 90.000,E1 98.106} C_DIS
LIN {X 0.136,Y -508.508,Z 1706.544,A 0.000,B 0.000,C 90.000,E1 97.871} C_DIS
LIN {X 0.204,Y -509.972,Z 1706.543,A 0.000,B 0.000,C 90.000,E1 97.644} C_DIS
LIN {X 0.153,Y -511.184,Z 1706.541,A 0.000,B 0.000,C 90.000,E1 97.409} C_DIS
LIN {X 0.037,Y -512.062,Z 1706.540,A 0.000,B 0.000,C 90.000,E1 97.182} C_DIS
LIN {X -0.116,Y -512.964,Z 1706.537,A 0.000,B 0.000,C 90.000,E1 96.720} C_DIS
LIN {X 0.245,Y -512.843,Z 1706.535,A 0.000,B 0.000,C 90.000,E1 96.201} C_DIS
LIN {X 0.100,Y -511.674,Z 1706.532,A 0.000,B 0.000,C 90.000,E1 95.739} C_DIS
LIN {X 0.003,Y -510.638,Z 1706.531,A 0.000,B 0.000,C 90.000,E1 95.511} C_DIS
LIN {X -0.046,Y -509.229,Z 1706.529,A 0.000,B 0.000,C 90.000,E1 95.277} C_DIS
LIN {X -0.114,Y -498.459,Z 1706.521,A 0.000,B 0.000,C 90.000,E1 93.841} C_DIS
LIN {X -0.043,Y -485.824,Z 1706.512,A 0.000,B 0.000,C 90.000,E1 92.121} C_DIS
LIN {X -0.036,Y -474.960,Z 1706.503,A 0.000,B 0.000,C 90.000,E1 90.630} C_DIS
LIN {X 0.041,Y -462.198,Z 1706.494,A 0.000,B 0.000,C 90.000,E1 88.854} C_DIS
LIN {X -0.133,Y -449.255,Z 1706.484,A 0.000,B 0.000,C 90.000,E1 87.078} C_DIS
LIN {X -0.092,Y -436.222,Z 1706.474,A 0.000,B 0.000,C 90.000,E1 85.241} C_DIS
LIN {X -0.122,Y -421.336,Z 1706.462,A 0.000,B 0.000,C 90.000,E1 83.109} C_DIS
LIN {X 0.075,Y -405.114,Z 1706.448,A 0.000,B 0.000,C 90.000,E1 80.622} C_DIS
LIN {X 0.031,Y -388.056,Z 1706.432,A 0.000,B 0.000,C 90.000,E1 77.825} C_DIS
LIN {X 0.100,Y -374.998,Z 1706.420,A 0.000,B 0.000,C 90.000,E1 75.519} C_DIS
LIN {X -0.034,Y -362.334,Z 1706.407,A 0.000,B 0.000,C 90.000,E1 73.196} C_DIS
LIN {X 0.008,Y -348.479,Z 1706.392,A 0.000,B 0.000,C 90.000,E1 70.496} C_DIS
LIN {X 0.132,Y -335.304,Z 1706.376,A 0.000,B 0.000,C 90.000,E1 67.720} C_DIS
LIN {X 0.029,Y -322.508,Z 1706.361,A 0.000,B 0.000,C 90.000,E1 64.921} C_DIS
LIN {X -0.002,Y -312.866,Z 1706.348,A 0.000,B 0.000,C 90.000,E1 62.692} C_DIS
LIN {X 0.080,Y -302.032,Z 1706.334,A 0.000,B 0.000,C 90.000,E1 60.078} C_DIS
LIN {X -0.057,Y -292.595,Z 1706.321,A 0.000,B 0.000,C 90.000,E1 57.788} C_DIS
LIN {X 0.028,Y -284.380,Z 1706.310,A 0.000,B 0.000,C 90.000,E1 55.754} C_DIS
LIN {X 0.041,Y -275.996,Z 1706.298,A 0.000,B 0.000,C 90.000,E1 53.703} C_DIS
LIN {X 0.138,Y -266.104,Z 1706.285,A 0.000,B 0.000,C 90.000,E1 51.251} C_DIS
LIN {X 0.147,Y -256.298,Z 1706.271,A 0.000,B 0.000,C 90.000,E1 48.771} C_DIS
LIN {X -0.080,Y -244.155,Z 1706.253,A 0.000,B 0.000,C 90.000,E1 45.567} C_DIS
LIN {X 0.048,Y -232.919,Z 1706.234,A 0.000,B 0.000,C 90.000,E1 42.204} C_DIS
LIN {X -0.026,Y -223.731,Z 1706.218,A 0.000,B 0.000,C 90.000,E1 39.197} C_DIS
LIN {X 0.080,Y -215.436,Z 1706.201,A 0.000,B 0.000,C 90.000,E1 36.091} C_DIS
LIN {X 0.081,Y -207.882,Z 1706.183,A 0.000,B 0.000,C 90.000,E1 32.959} C_DIS
LIN {X 0.021,Y -201.069,Z 1706.166,A 0.000,B 0.000,C 90.000,E1 29.795} C_DIS
LIN {X 0.025,Y -194.834,Z 1706.148,A 0.000,B 0.000,C 90.000,E1 26.565} C_DIS
LIN {X 0.047,Y -187.883,Z 1706.125,A 0.000,B 0.000,C 90.000,E1 22.461} C_DIS
LIN {X 0.035,Y -182.997,Z 1706.106,A 0.000,B 0.000,C 90.000,E1 19.141} C_DIS
LIN {X 0.014,Y -178.865,Z 1706.088,A 0.000,B 0.000,C 90.000,E1 15.788} C_DIS
LIN {X -0.028,Y -175.414,Z 1706.069,A 0.000,B 0.000,C 90.000,E1 12.411} C_DIS
LIN {X 0.060,Y -172.038,Z 1706.045,A 0.000,B 0.000,C 90.000,E1 8.106} C_DIS
LIN {X -0.078,Y -169.221,Z 1706.016,A 0.000,B 0.000,C 90.000,E1 2.980} C_DIS
LIN {X -0.003,Y -167.733,Z 1705.964,A 0.000,B 0.000,C 90.000,E1 353.451} C_DIS
LIN {X -0.030,Y -169.672,Z 1705.920,A 0.000,B 0.000,C 90.000,E1 345.644} C_DIS
LIN {X 0.081,Y -172.517,Z 1705.891,A 0.000,B 0.000,C 90.000,E1 340.423} C_DIS
LIN {X -0.055,Y -176.136,Z 1705.868,A 0.000,B 0.000,C 90.000,E1 336.177} C_DIS
LIN {X 0.029,Y -180.693,Z 1705.844,A 0.000,B 0.000,C 90.000,E1 331.897} C_DIS
LIN {X 0.006,Y -185.312,Z 1705.825,A 0.000,B 0.000,C 90.000,E1 328.535} C_DIS
LIN {X 0.086,Y -189.441,Z 1705.811,A 0.000,B 0.000,C 90.000,E1 326.008} C_DIS
LIN {X 0.037,Y -194.247,Z 1705.797,A 0.000,B 0.000,C 90.000,E1 323.543} C_DIS
LIN {X 0.038,Y -199.681,Z 1705.784,A 0.000,B 0.000,C 90.000,E1 321.090} C_DIS
LIN {X 0.129,Y -206.895,Z 1705.768,A 0.000,B 0.000,C 90.000,E1 318.243} C_DIS
LIN {X 0.069,Y -215.145,Z 1705.753,A 0.000,B 0.000,C 90.000,E1 315.486} C_DIS
LIN {X 0.041,Y -224.501,Z 1705.738,A 0.000,B 0.000,C 90.000,E1 312.771} C_DIS
LIN {X 0.128,Y -233.482,Z 1705.725,A 0.000,B 0.000,C 90.000,E1 310.458} C_DIS
LIN {X -0.065,Y -243.625,Z 1705.712,A 0.000,B 0.000,C 90.000,E1 308.257} C_DIS
LIN {X -0.094,Y -251.141,Z 1705.704,A 0.000,B 0.000,C 90.000,E1 306.790} C_DIS
LIN {X -0.055,Y -263.511,Z 1705.692,A 0.000,B 0.000,C 90.000,E1 304.612} C_DIS
LIN {X -0.043,Y -281.614,Z 1705.677,A 0.000,B 0.000,C 90.000,E1 301.799} C_DIS
LIN {X -0.002,Y -301.111,Z 1705.661,A 0.000,B 0.000,C 90.000,E1 299.077} C_DIS
LIN {X -0.135,Y -316.321,Z 1705.651,A 0.000,B 0.000,C 90.000,E1 297.129} C_DIS
LIN {X -0.179,Y -334.249,Z 1705.638,A 0.000,B 0.000,C 90.000,E1 294.899} C_DIS
LIN {X -0.091,Y -347.049,Z 1705.630,A 0.000,B 0.000,C 90.000,E1 293.334} C_DIS
LIN {X 0.068,Y -359.766,Z 1705.621,A 0.000,B 0.000,C 90.000,E1 291.791} C_DIS
LIN {X -0.016,Y -369.649,Z 1705.615,A 0.000,B 0.000,C 90.000,E1 290.610} C_DIS
LIN {X 0.133,Y -376.649,Z 1705.610,A 0.000,B 0.000,C 90.000,E1 289.704} C_DIS
LIN {X -0.011,Y -382.944,Z 1705.605,A 0.000,B 0.000,C 90.000,E1 288.852} C_DIS
LIN {X -0.117,Y -386.728,Z 1705.602,A 0.000,B 0.000,C 90.000,E1 288.290} C_DIS
LIN {X 0.045,Y -390.102,Z 1705.598,A 0.000,B 0.000,C 90.000,E1 287.692} C_DIS
LIN {X -0.142,Y -393.038,Z 1705.595,A 0.000,B 0.000,C 90.000,E1 287.149} C_DIS
LIN {X 0.121,Y -396.637,Z 1705.590,A 0.000,B 0.000,C 90.000,E1 286.260} C_DIS
LIN {X 0.039,Y -399.414,Z 1705.586,A 0.000,B 0.000,C 90.000,E1 285.426} C_DIS
LIN {X -0.101,Y -400.827,Z 1705.583,A 0.000,B 0.000,C 90.000,E1 284.883} C_DIS
LIN {X 0.054,Y -401.819,Z 1705.579,A 0.000,B 0.000,C 90.000,E1 284.300} C_DIS
LIN {X -0.168,Y -402.394,Z 1705.576,A 0.000,B 0.000,C 90.000,E1 283.772} C_DIS
LIN {X 0.100,Y -402.622,Z 1705.573,A 0.000,B 0.000,C 90.000,E1 283.175} C_DIS
LIN {X -0.114,Y -402.404,Z 1705.570,A 0.000,B 0.000,C 90.000,E1 282.647} C_DIS
LIN {X 0.067,Y -401.767,Z 1705.567,A 0.000,B 0.000,C 90.000,E1 282.063} C_DIS
LIN {X -0.145,Y -400.605,Z 1705.564,A 0.000,B 0.000,C 90.000,E1 281.535} C_DIS
LIN {X 0.031,Y -398.979,Z 1705.561,A 0.000,B 0.000,C 90.000,E1 280.950} C_DIS
LIN {X 0.197,Y -396.758,Z 1705.558,A 0.000,B 0.000,C 90.000,E1 280.366} C_DIS
LIN {X -0.111,Y -394.060,Z 1705.555,A 0.000,B 0.000,C 90.000,E1 279.849} C_DIS
LIN {X 0.081,Y -389.189,Z 1705.550,A 0.000,B 0.000,C 90.000,E1 278.973} C_DIS
LIN {X 0.202,Y -382.128,Z 1705.544,A 0.000,B 0.000,C 90.000,E1 277.814} C_DIS
LIN {X -0.148,Y -376.256,Z 1705.539,A 0.000,B 0.000,C 90.000,E1 277.004} C_DIS
LIN {X -0.174,Y -371.751,Z 1705.536,A 0.000,B 0.000,C 90.000,E1 276.429} C_DIS
LIN {X 0.142,Y -366.602,Z 1705.532,A 0.000,B 0.000,C 90.000,E1 275.796} C_DIS
LIN {X 0.130,Y -360.781,Z 1705.529,A 0.000,B 0.000,C 90.000,E1 275.220} C_DIS
LIN {X 0.142,Y -354.927,Z 1705.526,A 0.000,B 0.000,C 90.000,E1 274.702} C_DIS
LIN {X 0.020,Y -348.834,Z 1705.524,A 0.000,B 0.000,C 90.000,E1 274.245} C_DIS
LIN {X 0.120,Y -342.422,Z 1705.521,A 0.000,B 0.000,C 90.000,E1 273.784} C_DIS
LIN {X 0.116,Y -335.895,Z 1705.519,A 0.000,B 0.000,C 90.000,E1 273.383} C_DIS
LIN {X 0.086,Y -326.000,Z 1705.516,A 0.000,B 0.000,C 90.000,E1 272.865} C_DIS
LIN {X -0.004,Y -319.316,Z 1705.514,A 0.000,B 0.000,C 90.000,E1 272.579} C_DIS
LIN {X 0.089,Y -312.563,Z 1705.513,A 0.000,B 0.000,C 90.000,E1 272.293} C_DIS
LIN {X 0.075,Y -302.346,Z 1705.511,A 0.000,B 0.000,C 90.000,E1 271.949} C_DIS
LIN {X 0.047,Y -291.998,Z 1705.509,A 0.000,B 0.000,C 90.000,E1 271.661} C_DIS
LIN {X -0.040,Y -280.531,Z 1705.508,A 0.000,B 0.000,C 90.000,E1 271.432} C_DIS
LIN {X 0.121,Y -268.448,Z 1705.507,A 0.000,B 0.000,C 90.000,E1 271.203} C_DIS
LIN {X -0.103,Y -257.644,Z 1705.506,A 0.000,B 0.000,C 90.000,E1 271.146} C_DIS
LIN {X -0.035,Y -248.566,Z 1705.506,A 0.000,B 0.000,C 90.000,E1 271.088} C_DIS
LIN {X -0.048,Y -181.440,Z 1705.506,A 0.000,B 0.000,C 90.000,E1 271.088} C_DIS
LIN {X 0.004,Y -181.569,Z 1705.500,A 0.000,B 0.000,C 90.000,E1 270.057} C_DIS
LIN {X 0.007,Y -180.818,Z 1705.471,A 0.000,B 0.000,C 90.000,E1 264.837} C_DIS
LIN {X 0.083,Y -178.921,Z 1705.443,A 0.000,B 0.000,C 90.000,E1 259.746} C_DIS
LIN {X -0.008,Y -175.966,Z 1705.415,A 0.000,B 0.000,C 90.000,E1 254.685} C_DIS
LIN {X -0.060,Y -175.446,Z 1705.410,A 0.000,B 0.000,C 90.000,E1 253.850} C_DIS
LIN {X -0.051,Y -172.202,Z 1705.386,A 0.000,B 0.000,C 90.000,E1 249.571} C_DIS
LIN {X -0.073,Y -171.676,Z 1705.382,A 0.000,B 0.000,C 90.000,E1 248.720} C_DIS
LIN {X -0.082,Y -167.901,Z 1705.358,A 0.000,B 0.000,C 90.000,E1 244.409} C_DIS
LIN {X 0.085,Y -166.641,Z 1705.348,A 0.000,B 0.000,C 90.000,E1 242.615} C_DIS
LIN {X -0.008,Y -162.626,Z 1705.324,A 0.000,B 0.000,C 90.000,E1 238.280} C_DIS
LIN {X 0.051,Y -161.313,Z 1705.314,A 0.000,B 0.000,C 90.000,E1 236.501} C_DIS
LIN {X -0.040,Y -157.310,Z 1705.289,A 0.000,B 0.000,C 90.000,E1 232.110} C_DIS
LIN {X -0.106,Y -155.287,Z 1705.275,A 0.000,B 0.000,C 90.000,E1 229.461} C_DIS
LIN {X 0.041,Y -151.650,Z 1705.250,A 0.000,B 0.000,C 90.000,E1 224.919} C_DIS
LIN {X -0.022,Y -150.518,Z 1705.240,A 0.000,B 0.000,C 90.000,E1 223.137} C_DIS
LIN {X 0.001,Y -147.243,Z 1705.214,A 0.000,B 0.000,C 90.000,E1 218.588} C_DIS
LIN {X -0.034,Y -145.267,Z 1705.194,A 0.000,B 0.000,C 90.000,E1 214.945} C_DIS
LIN {X 0.000,Y -142.375,Z 1705.163,A 0.000,B 0.000,C 90.000,E1 209.411} C_DIS
LIN {X 0.049,Y -141.351,Z 1705.148,A 0.000,B 0.000,C 90.000,E1 206.616} C_DIS
LIN {X 0.033,Y -139.340,Z 1705.112,A 0.000,B 0.000,C 90.000,E1 200.120} C_DIS
LIN {X 0.083,Y -139.006,Z 1705.101,A 0.000,B 0.000,C 90.000,E1 198.236} C_DIS
LIN {X 0.039,Y -138.339,Z 1705.055,A 0.000,B 0.000,C 90.000,E1 189.849} C_DIS
LIN {X 0.062,Y -139.404,Z 1705.008,A 0.000,B 0.000,C 90.000,E1 181.432} C_DIS
LIN {X -0.024,Y -141.311,Z 1704.972,A 0.000,B 0.000,C 90.000,E1 174.951} C_DIS
LIN {X -0.067,Y -142.671,Z 1704.956,A 0.000,B 0.000,C 90.000,E1 172.186} C_DIS
LIN {X 0.054,Y -145.021,Z 1704.931,A 0.000,B 0.000,C 90.000,E1 167.521} C_DIS
LIN {X 0.012,Y -147.648,Z 1704.910,A 0.000,B 0.000,C 90.000,E1 163.866} C_DIS
LIN {X -0.053,Y -150.283,Z 1704.890,A 0.000,B 0.000,C 90.000,E1 160.242} C_DIS
LIN {X -0.040,Y -153.688,Z 1704.870,A 0.000,B 0.000,C 90.000,E1 156.613} C_DIS
LIN {X 0.015,Y -157.102,Z 1704.850,A 0.000,B 0.000,C 90.000,E1 152.999} C_DIS
LIN {X -0.047,Y -161.242,Z 1704.830,A 0.000,B 0.000,C 90.000,E1 149.459} C_DIS
LIN {X 0.038,Y -163.329,Z 1704.820,A 0.000,B 0.000,C 90.000,E1 147.661} C_DIS
LIN {X -0.091,Y -167.782,Z 1704.801,A 0.000,B 0.000,C 90.000,E1 144.196} C_DIS
LIN {X 0.061,Y -171.597,Z 1704.786,A 0.000,B 0.000,C 90.000,E1 141.537} C_DIS
LIN {X -0.009,Y -176.549,Z 1704.767,A 0.000,B 0.000,C 90.000,E1 138.119} C_DIS
LIN {X -0.016,Y -180.848,Z 1704.753,A 0.000,B 0.000,C 90.000,E1 135.567} C_DIS
LIN {X -0.033,Y -186.259,Z 1704.734,A 0.000,B 0.000,C 90.000,E1 132.204} C_DIS
LIN {X -0.096,Y -190.895,Z 1704.721,A 0.000,B 0.000,C 90.000,E1 129.725} C_DIS
LIN {X 0.095,Y -196.660,Z 1704.702,A 0.000,B 0.000,C 90.000,E1 126.377} C_DIS
LIN {X 0.013,Y -199.902,Z 1704.693,A 0.000,B 0.000,C 90.000,E1 124.771} C_DIS
LIN {X 0.045,Y -204.295,Z 1704.680,A 0.000,B 0.000,C 90.000,E1 122.339} C_DIS
LIN {X 0.026,Y -209.044,Z 1704.666,A 0.000,B 0.000,C 90.000,E1 119.951} C_DIS
LIN {X 0.006,Y -332.526,Z 1704.666,A 0.000,B 0.000,C 90.000,E1 119.951} C_DIS
LIN {X -0.096,Y -336.357,Z 1704.666,A 0.000,B 0.000,C 90.000,E1 119.873} C_DIS
LIN {X 0.098,Y -339.438,Z 1704.665,A 0.000,B 0.000,C 90.000,E1 119.667} C_DIS
LIN {X 0.054,Y -343.119,Z 1704.663,A 0.000,B 0.000,C 90.000,E1 119.333} C_DIS
LIN {X 0.010,Y -346.620,Z 1704.660,A 0.000,B 0.000,C 90.000,E1 118.821} C_DIS
LIN {X 0.174,Y -362.408,Z 1704.642,A 0.000,B 0.000,C 90.000,E1 115.463} C_DIS
LIN {X 0.056,Y -376.915,Z 1704.627,A 0.000,B 0.000,C 90.000,E1 112.823} C_DIS
LIN {X -0.112,Y -391.193,Z 1704.614,A 0.000,B 0.000,C 90.000,E1 110.536} C_DIS
LIN {X 0.173,Y -406.876,Z 1704.601,A 0.000,B 0.000,C 90.000,E1 108.236} C_DIS
LIN {X -0.177,Y -424.072,Z 1704.589,A 0.000,B 0.000,C 90.000,E1 106.079} C_DIS
LIN {X 0.183,Y -442.899,Z 1704.577,A 0.000,B 0.000,C 90.000,E1 103.883} C_DIS
LIN {X -0.019,Y -462.838,Z 1704.566,A 0.000,B 0.000,C 90.000,E1 101.883} C_DIS
LIN {X 0.033,Y -485.911,Z 1704.554,A 0.000,B 0.000,C 90.000,E1 99.792} C_DIS
LIN {X 0.231,Y -504.301,Z 1704.546,A 0.000,B 0.000,C 90.000,E1 98.276} C_DIS
LIN {X -0.065,Y -506.587,Z 1704.545,A 0.000,B 0.000,C 90.000,E1 98.106} C_DIS
LIN {X 0.212,Y -508.324,Z 1704.544,A 0.000,B 0.000,C 90.000,E1 97.871} C_DIS
LIN {X 0.089,Y -509.897,Z 1704.542,A 0.000,B 0.000,C 90.000,E1 97.644} C_DIS
LIN {X 0.033,Y -511.067,Z 1704.541,A 0.000,B 0.000,C 90.000,E1 97.409} C_DIS
LIN {X -0.129,Y -512.459,Z 1704.539,A 0.000,B 0.000,C 90.000,E1 96.947} C_DIS
LIN {X 0.223,Y -512.782,Z 1704.536,A 0.000,B 0.000,C 90.000,E1 96.429} C_DIS
LIN {X 0.076,Y -512.087,Z 1704.533,A 0.000,B 0.000,C 90.000,E1 95.967} C_DIS
LIN {X -0.121,Y -510.252,Z 1704.531,A 0.000,B 0.000,C 90.000,E1 95.511} C_DIS
LIN {X -0.171,Y -508.792,Z 1704.529,A 0.000,B 0.000,C 90.000,E1 95.277} C_DIS
LIN {X 0.133,Y -496.228,Z 1704.520,A 0.000,B 0.000,C 90.000,E1 93.555} C_DIS
LIN {X 0.159,Y -483.608,Z 1704.510,A 0.000,B 0.000,C 90.000,E1 91.835} C_DIS
LIN {X -0.056,Y -470.907,Z 1704.501,A 0.000,B 0.000,C 90.000,E1 90.115} C_DIS
LIN {X 0.152,Y -459.955,Z 1704.492,A 0.000,B 0.000,C 90.000,E1 88.568} C_DIS
LIN {X -0.048,Y -446.973,Z 1704.482,A 0.000,B 0.000,C 90.000,E1 86.788} C_DIS
LIN {X -0.046,Y -433.939,Z 1704.472,A 0.000,B 0.000,C 90.000,E1 84.951} C_DIS
LIN {X -0.030,Y -417.215,Z 1704.458,A 0.000,B 0.000,C 90.000,E1 82.534} C_DIS
LIN {X 0.121,Y -401.119,Z 1704.445,A 0.000,B 0.000,C 90.000,E1 80.038} C_DIS
LIN {X -0.001,Y -385.920,Z 1704.431,A 0.000,B 0.000,C 90.000,E1 77.521} C_DIS
LIN {X -0.065,Y -372.904,Z 1704.418,A 0.000,B 0.000,C 90.000,E1 75.227} C_DIS
LIN {X 0.096,Y -360.232,Z 1704.405,A 0.000,B 0.000,C 90.000,E1 72.851} C_DIS
LIN {X -0.148,Y -346.445,Z 1704.390,A 0.000,B 0.000,C 90.000,E1 70.188} C_DIS
LIN {X -0.070,Y -333.341,Z 1704.374,A 0.000,B 0.000,C 90.000,E1 67.411} C_DIS
LIN {X -0.141,Y -319.257,Z 1704.357,A 0.000,B 0.000,C 90.000,E1 64.280} C_DIS
LIN {X -0.036,Y -308.305,Z 1704.343,A 0.000,B 0.000,C 90.000,E1 61.691} C_DIS
LIN {X -0.076,Y -298.845,Z 1704.330,A 0.000,B 0.000,C 90.000,E1 59.410} C_DIS
LIN {X 0.122,Y -289.416,Z 1704.317,A 0.000,B 0.000,C 90.000,E1 57.041} C_DIS
LIN {X -0.092,Y -281.133,Z 1704.306,A 0.000,B 0.000,C 90.000,E1 55.055} C_DIS
LIN {X 0.028,Y -272.643,Z 1704.294,A 0.000,B 0.000,C 90.000,E1 52.970} C_DIS
LIN {X 0.058,Y -262.782,Z 1704.281,A 0.000,B 0.000,C 90.000,E1 50.517} C_DIS
LIN {X -0.009,Y -253.024,Z 1704.267,A 0.000,B 0.000,C 90.000,E1 48.038} C_DIS
LIN {X 0.019,Y -241.090,Z 1704.249,A 0.000,B 0.000,C 90.000,E1 44.757} C_DIS
LIN {X 0.067,Y -230.137,Z 1704.230,A 0.000,B 0.000,C 90.000,E1 41.391} C_DIS
LIN {X -0.004,Y -222.296,Z 1704.215,A 0.000,B 0.000,C 90.000,E1 38.749} C_DIS
LIN {X -0.056,Y -214.124,Z 1704.198,A 0.000,B 0.000,C 90.000,E1 35.678} C_DIS
LIN {X -0.079,Y -206.723,Z 1704.181,A 0.000,B 0.000,C 90.000,E1 32.546} C_DIS
LIN {X 0.008,Y -200.015,Z 1704.163,A 0.000,B 0.000,C 90.000,E1 29.333} C_DIS
LIN {X -0.014,Y -193.895,Z 1704.145,A 0.000,B 0.000,C 90.000,E1 26.104} C_DIS
LIN {X -0.007,Y -188.354,Z 1704.127,A 0.000,B 0.000,C 90.000,E1 22.823} C_DIS
LIN {X -0.009,Y -183.414,Z 1704.108,A 0.000,B 0.000,C 90.000,E1 19.504} C_DIS
LIN {X 0.031,Y -179.207,Z 1704.090,A 0.000,B 0.000,C 90.000,E1 16.134} C_DIS
LIN {X -0.048,Y -175.694,Z 1704.071,A 0.000,B 0.000,C 90.000,E1 12.771} C_DIS
LIN {X -0.085,Y -172.261,Z 1704.047,A 0.000,B 0.000,C 90.000,E1 8.511} C_DIS
LIN {X -0.041,Y -169.327,Z 1704.018,A 0.000,B 0.000,C 90.000,E1 3.326} C_DIS
LIN {X 0.001,Y -167.647,Z 1703.968,A 0.000,B 0.000,C 90.000,E1 354.318} C_DIS
LIN {X -0.063,Y -169.231,Z 1703.925,A 0.000,B 0.000,C 90.000,E1 346.520} C_DIS
LIN {X -0.063,Y -171.875,Z 1703.896,A 0.000,B 0.000,C 90.000,E1 341.329} C_DIS
LIN {X 0.043,Y -175.281,Z 1703.872,A 0.000,B 0.000,C 90.000,E1 336.997} C_DIS
LIN {X 0.019,Y -179.687,Z 1703.849,A 0.000,B 0.000,C 90.000,E1 332.743} C_DIS
LIN {X -0.027,Y -184.104,Z 1703.830,A 0.000,B 0.000,C 90.000,E1 329.380} C_DIS
LIN {X 0.072,Y -189.509,Z 1703.811,A 0.000,B 0.000,C 90.000,E1 326.008} C_DIS
LIN {X 0.025,Y -194.349,Z 1703.797,A 0.000,B 0.000,C 90.000,E1 323.543} C_DIS
LIN {X 0.026,Y -199.805,Z 1703.784,A 0.000,B 0.000,C 90.000,E1 321.090} C_DIS
LIN {X 0.121,Y -207.043,Z 1703.768,A 0.000,B 0.000,C 90.000,E1 318.243} C_DIS
LIN {X 0.064,Y -215.312,Z 1703.753,A 0.000,B 0.000,C 90.000,E1 315.486} C_DIS
LIN {X 0.039,Y -224.712,Z 1703.738,A 0.000,B 0.000,C 90.000,E1 312.771} C_DIS
LIN {X 0.132,Y -233.721,Z 1703.725,A 0.000,B 0.000,C 90.000,E1 310.458} C_DIS
LIN {X -0.059,Y -243.854,Z 1703.712,A 0.000,B 0.000,C 90.000,E1 308.257} C_DIS
LIN {X 0.124,Y -253.347,Z 1703.702,A 0.000,B 0.000,C 90.000,E1 306.377} C_DIS
LIN {X 0.000,Y -265.898,Z 1703.690,A 0.000,B 0.000,C 90.000,E1 304.246} C_DIS
LIN {X -0.077,Y -284.156,Z 1703.675,A 0.000,B 0.000,C 90.000,E1 301.465} C_DIS
LIN {X 0.030,Y -303.762,Z 1703.660,A 0.000,B 0.000,C 90.000,E1 298.743} C_DIS
LIN {X -0.104,Y -316.413,Z 1703.651,A 0.000,B 0.000,C 90.000,E1 297.129} C_DIS
LIN {X -0.098,Y -331.693,Z 1703.640,A 0.000,B 0.000,C 90.000,E1 295.207} C_DIS
LIN {X -0.076,Y -344.540,Z 1703.631,A 0.000,B 0.000,C 90.000,E1 293.643} C_DIS
LIN {X 0.163,Y -357.336,Z 1703.623,A 0.000,B 0.000,C 90.000,E1 292.078} C_DIS
LIN {X -0.076,Y -367.294,Z 1703.616,A 0.000,B 0.000,C 90.000,E1 290.918} C_DIS
LIN {X 0.170,Y -374.425,Z 1703.611,A 0.000,B 0.000,C 90.000,E1 289.993} C_DIS
LIN {X 0.010,Y -381.004,Z 1703.606,A 0.000,B 0.000,C 90.000,E1 289.141} C_DIS
LIN {X -0.102,Y -386.824,Z 1703.602,A 0.000,B 0.000,C 90.000,E1 288.290} C_DIS
LIN {X 0.095,Y -391.741,Z 1703.597,A 0.000,B 0.000,C 90.000,E1 287.402} C_DIS
LIN {X -0.079,Y -394.459,Z 1703.594,A 0.000,B 0.000,C 90.000,E1 286.858} C_DIS
LIN {X -0.184,Y -397.824,Z 1703.589,A 0.000,B 0.000,C 90.000,E1 286.024} C_DIS
LIN {X 0.058,Y -399.578,Z 1703.586,A 0.000,B 0.000,C 90.000,E1 285.426} C_DIS
LIN {X -0.081,Y -400.977,Z 1703.583,A 0.000,B 0.000,C 90.000,E1 284.883} C_DIS
LIN {X 0.075,Y -401.972,Z 1703.579,A 0.000,B 0.000,C 90.000,E1 284.300} C_DIS
LIN {X -0.147,Y -402.621,Z 1703.576,A 0.000,B 0.000,C 90.000,E1 283.772} C_DIS
LIN {X 0.123,Y -402.845,Z 1703.573,A 0.000,B 0.000,C 90.000,E1 283.175} C_DIS
LIN {X -0.089,Y -402.606,Z 1703.570,A 0.000,B 0.000,C 90.000,E1 282.647} C_DIS
LIN {X 0.093,Y -401.982,Z 1703.567,A 0.000,B 0.000,C 90.000,E1 282.063} C_DIS
LIN {X -0.119,Y -400.837,Z 1703.564,A 0.000,B 0.000,C 90.000,E1 281.535} C_DIS
LIN {X 0.058,Y -399.210,Z 1703.561,A 0.000,B 0.000,C 90.000,E1 280.950} C_DIS
LIN {X -0.155,Y -395.798,Z 1703.556,A 0.000,B 0.000,C 90.000,E1 280.141} C_DIS
LIN {X 0.062,Y -391.210,Z 1703.552,A 0.000,B 0.000,C 90.000,E1 279.265} C_DIS
LIN {X -0.170,Y -384.250,Z 1703.545,A 0.000,B 0.000,C 90.000,E1 278.163} C_DIS
LIN {X -0.127,Y -378.597,Z 1703.540,A 0.000,B 0.000,C 90.000,E1 277.296} C_DIS
LIN {X -0.139,Y -374.326,Z 1703.537,A 0.000,B 0.000,C 90.000,E1 276.720} C_DIS
LIN {X -0.173,Y -369.446,Z 1703.534,A 0.000,B 0.000,C 90.000,E1 276.144} C_DIS
LIN {X -0.164,Y -364.003,Z 1703.531,A 0.000,B 0.000,C 90.000,E1 275.568} C_DIS
LIN {X 0.056,Y -358.195,Z 1703.528,A 0.000,B 0.000,C 90.000,E1 274.992} C_DIS
LIN {X -0.155,Y -352.125,Z 1703.525,A 0.000,B 0.000,C 90.000,E1 274.531} C_DIS
LIN {X -0.129,Y -345.866,Z 1703.522,A 0.000,B 0.000,C 90.000,E1 274.069} C_DIS
LIN {X 0.099,Y -339.408,Z 1703.520,A 0.000,B 0.000,C 90.000,E1 273.612} C_DIS
LIN {X -0.100,Y -332.821,Z 1703.518,A 0.000,B 0.000,C 90.000,E1 273.269} C_DIS
LIN {X -0.043,Y -326.210,Z 1703.516,A 0.000,B 0.000,C 90.000,E1 272.922} C_DIS
LIN {X 0.021,Y -316.049,Z 1703.514,A 0.000,B 0.000,C 90.000,E1 272.465} C_DIS
LIN {X -0.122,Y -305.791,Z 1703.512,A 0.000,B 0.000,C 90.000,E1 272.121} C_DIS
LIN {X 0.048,Y -295.395,Z 1703.510,A 0.000,B 0.000,C 90.000,E1 271.776} C_DIS
LIN {X -0.107,Y -284.599,Z 1703.508,A 0.000,B 0.000,C 90.000,E1 271.547} C_DIS
LIN {X -0.042,Y -272.548,Z 1703.507,A 0.000,B 0.000,C 90.000,E1 271.318} C_DIS
LIN {X -0.090,Y -262.400,Z 1703.507,A 0.000,B 0.000,C 90.000,E1 271.203} C_DIS
LIN {X 0.100,Y -250.613,Z 1703.506,A 0.000,B 0.000,C 90.000,E1 271.088} C_DIS
LIN {X 0.051,Y -181.433,Z 1703.506,A 0.000,B 0.000,C 90.000,E1 271.088} C_DIS
LIN {X 0.061,Y -181.571,Z 1703.500,A 0.000,B 0.000,C 90.000,E1 270.057} C_DIS
LIN {X 0.063,Y -180.823,Z 1703.471,A 0.000,B 0.000,C 90.000,E1 264.837} C_DIS
LIN {X -0.037,Y -178.928,Z 1703.443,A 0.000,B 0.000,C 90.000,E1 259.803} C_DIS
LIN {X 0.002,Y -175.975,Z 1703.415,A 0.000,B 0.000,C 90.000,E1 254.700} C_DIS
LIN {X -0.053,Y -175.462,Z 1703.410,A 0.000,B 0.000,C 90.000,E1 253.866} C_DIS
LIN {X 0.004,Y -172.212,Z 1703.386,A 0.000,B 0.000,C 90.000,E1 249.571} C_DIS
LIN {X -0.019,Y -171.688,Z 1703.382,A 0.000,B 0.000,C 90.000,E1 248.720} C_DIS
LIN {X -0.028,Y -167.915,Z 1703.358,A 0.000,B 0.000,C 90.000,E1 244.409} C_DIS
LIN {X -0.010,Y -166.657,Z 1703.348,A 0.000,B 0.000,C 90.000,E1 242.666} C_DIS
LIN {X 0.045,Y -162.640,Z 1703.324,A 0.000,B 0.000,C 90.000,E1 238.280} C_DIS
LIN {X -0.030,Y -161.329,Z 1703.314,A 0.000,B 0.000,C 90.000,E1 236.548} C_DIS
LIN {X 0.012,Y -157.324,Z 1703.290,A 0.000,B 0.000,C 90.000,E1 232.110} C_DIS
LIN {X -0.055,Y -155.305,Z 1703.275,A 0.000,B 0.000,C 90.000,E1 229.461} C_DIS
LIN {X -0.016,Y -151.663,Z 1703.250,A 0.000,B 0.000,C 90.000,E1 224.960} C_DIS
LIN {X 0.028,Y -150.530,Z 1703.240,A 0.000,B 0.000,C 90.000,E1 223.137} C_DIS
LIN {X -0.042,Y -147.255,Z 1703.214,A 0.000,B 0.000,C 90.000,E1 218.624} C_DIS
LIN {X 0.015,Y -145.281,Z 1703.194,A 0.000,B 0.000,C 90.000,E1 214.945} C_DIS
LIN {X 0.049,Y -142.383,Z 1703.163,A 0.000,B 0.000,C 90.000,E1 209.411} C_DIS
LIN {X -0.028,Y -141.360,Z 1703.148,A 0.000,B 0.000,C 90.000,E1 206.668} C_DIS
LIN {X -0.050,Y -139.342,Z 1703.112,A 0.000,B 0.000,C 90.000,E1 200.174} C_DIS
LIN {X -0.044,Y -139.012,Z 1703.102,A 0.000,B 0.000,C 90.000,E1 198.308} C_DIS
LIN {X -0.049,Y -138.341,Z 1703.055,A 0.000,B 0.000,C 90.000,E1 189.905} C_DIS
LIN {X -0.029,Y -139.399,Z 1703.008,A 0.000,B 0.000,C 90.000,E1 181.489} C_DIS
LIN {X 0.024,Y -141.302,Z 1702.972,A 0.000,B 0.000,C 90.000,E1 174.951} C_DIS
LIN {X -0.019,Y -142.663,Z 1702.957,A 0.000,B 0.000,C 90.000,E1 172.186} C_DIS
LIN {X -0.069,Y -145.009,Z 1702.931,A 0.000,B 0.000,C 90.000,E1 167.589} C_DIS
LIN {X -0.080,Y -147.637,Z 1702.911,A 0.000,B 0.000,C 90.000,E1 163.921} C_DIS
LIN {X -0.003,Y -150.267,Z 1702.890,A 0.000,B 0.000,C 90.000,E1 160.242} C_DIS
LIN {X 0.011,Y -153.668,Z 1702.870,A 0.000,B 0.000,C 90.000,E1 156.613} C_DIS
LIN {X 0.067,Y -157.082,Z 1702.850,A 0.000,B 0.000,C 90.000,E1 152.999} C_DIS
LIN {X 0.006,Y -161.218,Z 1702.830,A 0.000,B 0.000,C 90.000,E1 149.459} C_DIS
LIN {X -0.047,Y -163.307,Z 1702.821,A 0.000,B 0.000,C 90.000,E1 147.709} C_DIS
LIN {X -0.037,Y -167.757,Z 1702.801,A 0.000,B 0.000,C 90.000,E1 144.196} C_DIS
LIN {X -0.019,Y -171.573,Z 1702.786,A 0.000,B 0.000,C 90.000,E1 141.582} C_DIS
LIN {X -0.084,Y -176.520,Z 1702.767,A 0.000,B 0.000,C 90.000,E1 138.162} C_DIS
LIN {X 0.040,Y -180.819,Z 1702.753,A 0.000,B 0.000,C 90.000,E1 135.567} C_DIS
LIN {X 0.025,Y -186.228,Z 1702.734,A 0.000,B 0.000,C 90.000,E1 132.204} C_DIS
LIN {X -0.037,Y -190.865,Z 1702.721,A 0.000,B 0.000,C 90.000,E1 129.725} C_DIS
LIN {X -0.004,Y -196.627,Z 1702.702,A 0.000,B 0.000,C 90.000,E1 126.423} C_DIS
LIN {X -0.091,Y -199.866,Z 1702.693,A 0.000,B 0.000,C 90.000,E1 124.818} C_DIS
LIN {X 0.105,Y -204.264,Z 1702.680,A 0.000,B 0.000,C 90.000,E1 122.339} C_DIS
LIN {X -0.037,Y -208.975,Z 1702.667,A 0.000,B 0.000,C 90.000,E1 120.001} C_DIS
LIN {X -0.100,Y -332.640,Z 1702.667,A 0.000,B 0.000,C 90.000,E1 120.001} C_DIS
LIN {X -0.073,Y -336.861,Z 1702.666,A 0.000,B 0.000,C 90.000,E1 119.873} C_DIS
LIN {X -0.093,Y -340.139,Z 1702.665,A 0.000,B 0.000,C 90.000,E1 119.667} C_DIS
LIN {X -0.084,Y -343.816,Z 1702.663,A 0.000,B 0.000,C 90.000,E1 119.283} C_DIS
LIN {X -0.077,Y -345.720,Z 1702.661,A 0.000,B 0.000,C 90.000,E1 118.999} C_DIS
LIN {X 0.066,Y -347.214,Z 1702.659,A 0.000,B 0.000,C 90.000,E1 118.693} C_DIS
LIN {X -0.001,Y -359.941,Z 1702.644,A 0.000,B 0.000,C 90.000,E1 115.976} C_DIS
LIN {X -0.191,Y -374.165,Z 1702.630,A 0.000,B 0.000,C 90.000,E1 113.334} C_DIS
LIN {X 0.077,Y -388.171,Z 1702.617,A 0.000,B 0.000,C 90.000,E1 110.972} C_DIS
LIN {X -0.085,Y -403.561,Z 1702.604,A 0.000,B 0.000,C 90.000,E1 108.725} C_DIS
LIN {X 0.003,Y -420.441,Z 1702.592,A 0.000,B 0.000,C 90.000,E1 106.496} C_DIS
LIN {X -0.146,Y -438.926,Z 1702.580,A 0.000,B 0.000,C 90.000,E1 104.356} C_DIS
LIN {X -0.183,Y -458.736,Z 1702.568,A 0.000,B 0.000,C 90.000,E1 102.299} C_DIS
LIN {X 0.122,Y -479.120,Z 1702.558,A 0.000,B 0.000,C 90.000,E1 100.366} C_DIS
LIN {X 0.033,Y -505.216,Z 1702.546,A 0.000,B 0.000,C 90.000,E1 98.219} C_DIS
LIN {X -0.089,Y -508.835,Z 1702.543,A 0.000,B 0.000,C 90.000,E1 97.814} C_DIS
LIN {X -0.217,Y -510.220,Z 1702.542,A 0.000,B 0.000,C 90.000,E1 97.587} C_DIS
LIN {X 0.230,Y -511.240,Z 1702.541,A 0.000,B 0.000,C 90.000,E1 97.296} C_DIS
LIN {X 0.071,Y -512.378,Z 1702.538,A 0.000,B 0.000,C 90.000,E1 96.834} C_DIS
LIN {X -0.083,Y -512.476,Z 1702.535,A 0.000,B 0.000,C 90.000,E1 96.372} C_DIS
LIN {X -0.231,Y -511.545,Z 1702.533,A 0.000,B 0.000,C 90.000,E1 95.910} C_DIS
LIN {X 0.129,Y -509.415,Z 1702.530,A 0.000,B 0.000,C 90.000,E1 95.391} C_DIS
LIN {X -0.242,Y -502.423,Z 1702.525,A 0.000,B 0.000,C 90.000,E1 94.473} C_DIS
LIN {X -0.066,Y -489.823,Z 1702.515,A 0.000,B 0.000,C 90.000,E1 92.751} C_DIS
LIN {X -0.159,Y -477.143,Z 1702.506,A 0.000,B 0.000,C 90.000,E1 91.031} C_DIS
LIN {X -0.040,Y -464.458,Z 1702.496,A 0.000,B 0.000,C 90.000,E1 89.255} C_DIS
LIN {X 0.067,Y -453.383,Z 1702.487,A 0.000,B 0.000,C 90.000,E1 87.707} C_DIS
LIN {X 0.196,Y -440.380,Z 1702.477,A 0.000,B 0.000,C 90.000,E1 85.869} C_DIS
LIN {X 0.045,Y -427.258,Z 1702.467,A 0.000,B 0.000,C 90.000,E1 84.033} C_DIS
LIN {X -0.008,Y -410.725,Z 1702.453,A 0.000,B 0.000,C 90.000,E1 81.602} C_DIS
LIN {X 0.184,Y -389.885,Z 1702.435,A 0.000,B 0.000,C 90.000,E1 78.229} C_DIS
LIN {X -0.160,Y -376.733,Z 1702.422,A 0.000,B 0.000,C 90.000,E1 75.992} C_DIS
LIN {X 0.105,Y -363.933,Z 1702.409,A 0.000,B 0.000,C 90.000,E1 73.614} C_DIS
LIN {X 0.186,Y -349.933,Z 1702.394,A 0.000,B 0.000,C 90.000,E1 70.913} C_DIS
LIN {X -0.089,Y -335.232,Z 1702.377,A 0.000,B 0.000,C 90.000,E1 67.901} C_DIS
LIN {X 0.112,Y -322.460,Z 1702.361,A 0.000,B 0.000,C 90.000,E1 65.049} C_DIS
LIN {X 0.140,Y -311.468,Z 1702.347,A 0.000,B 0.000,C 90.000,E1 62.487} C_DIS
LIN {X -0.106,Y -302.019,Z 1702.335,A 0.000,B 0.000,C 90.000,E1 60.255} C_DIS
LIN {X 0.018,Y -292.566,Z 1702.322,A 0.000,B 0.000,C 90.000,E1 57.916} C_DIS
LIN {X 0.105,Y -284.380,Z 1702.311,A 0.000,B 0.000,C 90.000,E1 55.881} C_DIS
LIN {X -0.045,Y -275.984,Z 1702.299,A 0.000,B 0.000,C 90.000,E1 53.863} C_DIS
LIN {X -0.081,Y -264.632,Z 1702.284,A 0.000,B 0.000,C 90.000,E1 51.090} C_DIS
LIN {X -0.097,Y -254.849,Z 1702.270,A 0.000,B 0.000,C 90.000,E1 48.609} C_DIS
LIN {X -0.002,Y -242.771,Z 1702.252,A 0.000,B 0.000,C 90.000,E1 45.324} C_DIS
LIN {X -0.038,Y -232.875,Z 1702.235,A 0.000,B 0.000,C 90.000,E1 42.366} C_DIS
LIN {X 0.034,Y -223.727,Z 1702.219,A 0.000,B 0.000,C 90.000,E1 39.322} C_DIS
LIN {X 0.006,Y -215.473,Z 1702.201,A 0.000,B 0.000,C 90.000,E1 36.251} C_DIS
LIN {X 0.131,Y -207.930,Z 1702.184,A 0.000,B 0.000,C 90.000,E1 33.086} C_DIS
LIN {X 0.067,Y -201.135,Z 1702.166,A 0.000,B 0.000,C 90.000,E1 29.922} C_DIS
LIN {X -0.103,Y -194.903,Z 1702.148,A 0.000,B 0.000,C 90.000,E1 26.744} C_DIS
LIN {X -0.065,Y -189.292,Z 1702.130,A 0.000,B 0.000,C 90.000,E1 23.462} C_DIS
LIN {X 0.030,Y -184.215,Z 1702.112,A 0.000,B 0.000,C 90.000,E1 20.120} C_DIS
LIN {X -0.054,Y -178.917,Z 1702.089,A 0.000,B 0.000,C 90.000,E1 15.953} C_DIS
LIN {X 0.031,Y -175.459,Z 1702.070,A 0.000,B 0.000,C 90.000,E1 12.535} C_DIS
LIN {X -0.018,Y -172.085,Z 1702.046,A 0.000,B 0.000,C 90.000,E1 8.276} C_DIS
LIN {X 0.011,Y -169.200,Z 1702.017,A 0.000,B 0.000,C 90.000,E1 3.094} C_DIS
LIN {X 0.000,Y -167.576,Z 1701.968,A 0.000,B 0.000,C 90.000,E1 354.318} C_DIS
LIN {X 0.095,Y -169.164,Z 1701.925,A 0.000,B 0.000,C 90.000,E1 346.464} C_DIS
LIN {X 0.091,Y -171.805,Z 1701.896,A 0.000,B 0.000,C 90.000,E1 341.275} C_DIS
LIN {X 0.031,Y -175.233,Z 1701.872,A 0.000,B 0.000,C 90.000,E1 336.997} C_DIS
LIN {X 0.006,Y -179.690,Z 1701.849,A 0.000,B 0.000,C 90.000,E1 332.743} C_DIS
LIN {X 0.119,Y -184.130,Z 1701.830,A 0.000,B 0.000,C 90.000,E1 329.331} C_DIS
LIN {X 0.077,Y -188.114,Z 1701.816,A 0.000,B 0.000,C 90.000,E1 326.834} C_DIS
LIN {X 0.049,Y -192.766,Z 1701.802,A 0.000,B 0.000,C 90.000,E1 324.356} C_DIS
LIN {X 0.017,Y -198.034,Z 1701.788,A 0.000,B 0.000,C 90.000,E1 321.904} C_DIS
LIN {X -0.064,Y -205.022,Z 1701.773,A 0.000,B 0.000,C 90.000,E1 319.094} C_DIS
LIN {X -0.021,Y -212.987,Z 1701.757,A 0.000,B 0.000,C 90.000,E1 316.296} C_DIS
LIN {X 0.051,Y -222.127,Z 1701.742,A 0.000,B 0.000,C 90.000,E1 313.542} C_DIS
LIN {X 0.092,Y -230.839,Z 1701.729,A 0.000,B 0.000,C 90.000,E1 311.229} C_DIS
LIN {X -0.001,Y -240.572,Z 1701.717,A 0.000,B 0.000,C 90.000,E1 308.991} C_DIS
LIN {X -0.064,Y -247.767,Z 1701.708,A 0.000,B 0.000,C 90.000,E1 307.523} C_DIS
LIN {X 0.063,Y -259.653,Z 1701.696,A 0.000,B 0.000,C 90.000,E1 305.311} C_DIS
LIN {X -0.018,Y -277.297,Z 1701.681,A 0.000,B 0.000,C 90.000,E1 302.498} C_DIS
LIN {X 0.067,Y -296.414,Z 1701.665,A 0.000,B 0.000,C 90.000,E1 299.745} C_DIS
LIN {X -0.114,Y -313.986,Z 1701.652,A 0.000,B 0.000,C 90.000,E1 297.462} C_DIS
LIN {X -0.150,Y -329.181,Z 1701.642,A 0.000,B 0.000,C 90.000,E1 295.540} C_DIS
LIN {X 0.041,Y -341.932,Z 1701.633,A 0.000,B 0.000,C 90.000,E1 293.951} C_DIS
LIN {X -0.203,Y -357.290,Z 1701.623,A 0.000,B 0.000,C 90.000,E1 292.153} C_DIS
LIN {X 0.015,Y -367.249,Z 1701.616,A 0.000,B 0.000,C 90.000,E1 290.918} C_DIS
LIN {X -0.217,Y -374.386,Z 1701.611,A 0.000,B 0.000,C 90.000,E1 290.066} C_DIS
LIN {X 0.104,Y -380.979,Z 1701.606,A 0.000,B 0.000,C 90.000,E1 289.141} C_DIS
LIN {X -0.130,Y -386.842,Z 1701.602,A 0.000,B 0.000,C 90.000,E1 288.308} C_DIS
LIN {X 0.156,Y -390.252,Z 1701.598,A 0.000,B 0.000,C 90.000,E1 287.692} C_DIS
LIN {X 0.017,Y -394.554,Z 1701.594,A 0.000,B 0.000,C 90.000,E1 286.858} C_DIS
LIN {X -0.086,Y -397.939,Z 1701.589,A 0.000,B 0.000,C 90.000,E1 286.024} C_DIS
LIN {X 0.158,Y -399.701,Z 1701.586,A 0.000,B 0.000,C 90.000,E1 285.426} C_DIS
LIN {X -0.084,Y -401.132,Z 1701.583,A 0.000,B 0.000,C 90.000,E1 284.898} C_DIS
LIN {X 0.176,Y -402.180,Z 1701.580,A 0.000,B 0.000,C 90.000,E1 284.300} C_DIS
LIN {X -0.044,Y -402.803,Z 1701.576,A 0.000,B 0.000,C 90.000,E1 283.772} C_DIS
LIN {X 0.226,Y -403.026,Z 1701.573,A 0.000,B 0.000,C 90.000,E1 283.175} C_DIS
LIN {X 0.015,Y -402.867,Z 1701.570,A 0.000,B 0.000,C 90.000,E1 282.647} C_DIS
LIN {X 0.199,Y -402.195,Z 1701.567,A 0.000,B 0.000,C 90.000,E1 282.063} C_DIS
LIN {X -0.012,Y -401.128,Z 1701.564,A 0.000,B 0.000,C 90.000,E1 281.535} C_DIS
LIN {X 0.167,Y -399.498,Z 1701.561,A 0.000,B 0.000,C 90.000,E1 280.950} C_DIS
LIN {X -0.055,Y -397.402,Z 1701.558,A 0.000,B 0.000,C 90.000,E1 280.423} C_DIS
LIN {X 0.035,Y -394.701,Z 1701.555,A 0.000,B 0.000,C 90.000,E1 279.849} C_DIS
LIN {X -0.154,Y -389.920,Z 1701.550,A 0.000,B 0.000,C 90.000,E1 279.029} C_DIS
LIN {X -0.020,Y -382.800,Z 1701.544,A 0.000,B 0.000,C 90.000,E1 277.871} C_DIS
LIN {X 0.011,Y -376.849,Z 1701.539,A 0.000,B 0.000,C 90.000,E1 277.004} C_DIS
LIN {X -0.013,Y -372.235,Z 1701.536,A 0.000,B 0.000,C 90.000,E1 276.429} C_DIS
LIN {X -0.061,Y -367.019,Z 1701.532,A 0.000,B 0.000,C 90.000,E1 275.853} C_DIS
LIN {X -0.039,Y -361.212,Z 1701.529,A 0.000,B 0.000,C 90.000,E1 275.277} C_DIS
LIN {X -0.080,Y -355.128,Z 1701.526,A 0.000,B 0.000,C 90.000,E1 274.759} C_DIS
LIN {X 0.154,Y -348.888,Z 1701.524,A 0.000,B 0.000,C 90.000,E1 274.245} C_DIS
LIN {X -0.007,Y -342.530,Z 1701.521,A 0.000,B 0.000,C 90.000,E1 273.841} C_DIS
LIN {X 0.028,Y -335.951,Z 1701.519,A 0.000,B 0.000,C 90.000,E1 273.440} C_DIS
LIN {X 0.088,Y -326.234,Z 1701.516,A 0.000,B 0.000,C 90.000,E1 272.922} C_DIS
LIN {X -0.132,Y -316.183,Z 1701.514,A 0.000,B 0.000,C 90.000,E1 272.522} C_DIS
LIN {X 0.029,Y -305.863,Z 1701.512,A 0.000,B 0.000,C 90.000,E1 272.121} C_DIS
LIN {X -0.126,Y -295.449,Z 1701.510,A 0.000,B 0.000,C 90.000,E1 271.833} C_DIS
LIN {X 0.092,Y -288.157,Z 1701.509,A 0.000,B 0.000,C 90.000,E1 271.604} C_DIS
LIN {X 0.080,Y -276.250,Z 1701.508,A 0.000,B 0.000,C 90.000,E1 271.375} C_DIS
LIN {X 0.001,Y -262.039,Z 1701.507,A 0.000,B 0.000,C 90.000,E1 271.203} C_DIS
LIN {X -0.009,Y -251.364,Z 1701.506,A 0.000,B 0.000,C 90.000,E1 271.146} C_DIS
LIN {X -0.030,Y -181.426,Z 1701.506,A 0.000,B 0.000,C 90.000,E1 271.146} C_DIS
LIN {X 0.091,Y -181.581,Z 1701.501,A 0.000,B 0.000,C 90.000,E1 270.229} C_DIS
LIN {X 0.080,Y -180.896,Z 1701.473,A 0.000,B 0.000,C 90.000,E1 265.179} C_DIS
LIN {X -0.092,Y -179.842,Z 1701.459,A 0.000,B 0.000,C 90.000,E1 262.704} C_DIS
LIN {X -0.035,Y -179.026,Z 1701.445,A 0.000,B 0.000,C 90.000,E1 260.151} C_DIS
LIN {X 0.027,Y -178.671,Z 1701.441,A 0.000,B 0.000,C 90.000,E1 259.285} C_DIS
LIN {X -0.037,Y -175.721,Z 1701.412,A 0.000,B 0.000,C 90.000,E1 254.212} C_DIS
LIN {X -0.020,Y -172.438,Z 1701.388,A 0.000,B 0.000,C 90.000,E1 249.934} C_DIS
LIN {X -0.065,Y -171.267,Z 1701.379,A 0.000,B 0.000,C 90.000,E1 248.230} C_DIS
LIN {X -0.019,Y -167.537,Z 1701.355,A 0.000,B 0.000,C 90.000,E1 243.896} C_DIS
LIN {X -0.005,Y -166.154,Z 1701.345,A 0.000,B 0.000,C 90.000,E1 242.153} C_DIS
LIN {X -0.015,Y -162.930,Z 1701.326,A 0.000,B 0.000,C 90.000,E1 238.663} C_DIS
LIN {X -0.036,Y -161.602,Z 1701.316,A 0.000,B 0.000,C 90.000,E1 236.914} C_DIS
LIN {X -0.060,Y -159.126,Z 1701.301,A 0.000,B 0.000,C 90.000,E1 234.276} C_DIS
LIN {X -0.050,Y -155.648,Z 1701.277,A 0.000,B 0.000,C 90.000,E1 229.828} C_DIS
LIN {X 0.002,Y -151.919,Z 1701.252,A 0.000,B 0.000,C 90.000,E1 225.324} C_DIS
LIN {X 0.018,Y -150.154,Z 1701.237,A 0.000,B 0.000,C 90.000,E1 222.609} C_DIS
LIN {X -0.062,Y -146.936,Z 1701.212,A 0.000,B 0.000,C 90.000,E1 218.096} C_DIS
LIN {X 0.046,Y -145.523,Z 1701.196,A 0.000,B 0.000,C 90.000,E1 215.311} C_DIS
LIN {X 0.039,Y -142.923,Z 1701.171,A 0.000,B 0.000,C 90.000,E1 210.718} C_DIS
LIN {X -0.034,Y -141.545,Z 1701.150,A 0.000,B 0.000,C 90.000,E1 207.052} C_DIS
LIN {X -0.045,Y -139.403,Z 1701.114,A 0.000,B 0.000,C 90.000,E1 200.556} C_DIS
LIN {X 0.009,Y -139.121,Z 1701.104,A 0.000,B 0.000,C 90.000,E1 198.671} C_DIS
LIN {X 0.040,Y -138.352,Z 1701.057,A 0.000,B 0.000,C 90.000,E1 190.254} C_DIS
LIN {X 0.031,Y -139.502,Z 1701.005,A 0.000,B 0.000,C 90.000,E1 180.917} C_DIS
LIN {X -0.029,Y -141.133,Z 1700.974,A 0.000,B 0.000,C 90.000,E1 175.355} C_DIS
LIN {X -0.075,Y -142.514,Z 1700.959,A 0.000,B 0.000,C 90.000,E1 172.591} C_DIS
LIN {X 0.012,Y -144.773,Z 1700.933,A 0.000,B 0.000,C 90.000,E1 167.937} C_DIS
LIN {X -0.039,Y -147.387,Z 1700.913,A 0.000,B 0.000,C 90.000,E1 164.283} C_DIS
LIN {X 0.023,Y -150.717,Z 1700.887,A 0.000,B 0.000,C 90.000,E1 159.699} C_DIS
LIN {X -0.037,Y -154.198,Z 1700.867,A 0.000,B 0.000,C 90.000,E1 156.102} C_DIS
LIN {X 0.033,Y -157.638,Z 1700.847,A 0.000,B 0.000,C 90.000,E1 152.487} C_DIS
LIN {X -0.020,Y -161.896,Z 1700.827,A 0.000,B 0.000,C 90.000,E1 148.948} C_DIS
LIN {X 0.089,Y -166.086,Z 1700.808,A 0.000,B 0.000,C 90.000,E1 145.388} C_DIS
LIN {X 0.087,Y -171.095,Z 1700.789,A 0.000,B 0.000,C 90.000,E1 141.904} C_DIS
LIN {X 0.008,Y -175.968,Z 1700.769,A 0.000,B 0.000,C 90.000,E1 138.485} C_DIS
LIN {X 0.121,Y -180.213,Z 1700.755,A 0.000,B 0.000,C 90.000,E1 135.891} C_DIS
LIN {X 0.096,Y -185.628,Z 1700.736,A 0.000,B 0.000,C 90.000,E1 132.528} C_DIS
LIN {X -0.119,Y -190.224,Z 1700.723,A 0.000,B 0.000,C 90.000,E1 130.092} C_DIS
LIN {X 0.041,Y -197.553,Z 1700.700,A 0.000,B 0.000,C 90.000,E1 125.931} C_DIS
LIN {X -0.034,Y -200.818,Z 1700.691,A 0.000,B 0.000,C 90.000,E1 124.326} C_DIS
LIN {X 0.052,Y -206.712,Z 1700.673,A 0.000,B 0.000,C 90.000,E1 121.082} C_DIS
LIN {X 0.110,Y -208.891,Z 1700.667,A 0.000,B 0.000,C 90.000,E1 120.001} C_DIS
LIN {X 0.130,Y -331.762,Z 1700.667,A 0.000,B 0.000,C 90.000,E1 120.001} C_DIS
LIN {X 0.040,Y -333.177,Z 1700.667,A 0.000,B 0.000,C 90.000,E1 120.001} C_DIS
LIN {X 0.059,Y -339.050,Z 1700.665,A 0.000,B 0.000,C 90.000,E1 119.745} C_DIS
LIN {X 0.079,Y -341.948,Z 1700.664,A 0.000,B 0.000,C 90.000,E1 119.489} C_DIS
LIN {X 0.044,Y -345.632,Z 1700.661,A 0.000,B 0.000,C 90.000,E1 118.999} C_DIS
LIN {X 0.196,Y -348.577,Z 1700.658,A 0.000,B 0.000,C 90.000,E1 118.359} C_DIS
LIN {X 0.011,Y -361.454,Z 1700.643,A 0.000,B 0.000,C 90.000,E1 115.668} C_DIS
LIN {X -0.131,Y -375.856,Z 1700.628,A 0.000,B 0.000,C 90.000,E1 113.025} C_DIS
LIN {X 0.183,Y -390.032,Z 1700.615,A 0.000,B 0.000,C 90.000,E1 110.663} C_DIS
LIN {X 0.069,Y -405.607,Z 1700.602,A 0.000,B 0.000,C 90.000,E1 108.417} C_DIS
LIN {X 0.089,Y -422.685,Z 1700.590,A 0.000,B 0.000,C 90.000,E1 106.205} C_DIS
LIN {X 0.006,Y -441.385,Z 1700.578,A 0.000,B 0.000,C 90.000,E1 104.064} C_DIS
LIN {X 0.148,Y -461.280,Z 1700.567,A 0.000,B 0.000,C 90.000,E1 102.007} C_DIS
LIN {X 0.191,Y -484.310,Z 1700.555,A 0.000,B 0.000,C 90.000,E1 99.905} C_DIS
LIN {X 0.002,Y -505.195,Z 1700.546,A 0.000,B 0.000,C 90.000,E1 98.219} C_DIS
LIN {X 0.196,Y -507.152,Z 1700.545,A 0.000,B 0.000,C 90.000,E1 97.992} C_DIS
LIN {X 0.139,Y -508.899,Z 1700.543,A 0.000,B 0.000,C 90.000,E1 97.757} C_DIS
LIN {X 0.013,Y -510.206,Z 1700.542,A 0.000,B 0.000,C 90.000,E1 97.530} C_DIS
LIN {X -0.152,Y -511.811,Z 1700.539,A 0.000,B 0.000,C 90.000,E1 97.068} C_DIS
LIN {X 0.199,Y -512.318,Z 1700.536,A 0.000,B 0.000,C 90.000,E1 96.549} C_DIS
LIN {X 0.051,Y -511.811,Z 1700.534,A 0.000,B 0.000,C 90.000,E1 96.087} C_DIS
LIN {X -0.096,Y -510.202,Z 1700.531,A 0.000,B 0.000,C 90.000,E1 95.625} C_DIS
LIN {X -0.146,Y -508.893,Z 1700.530,A 0.000,B 0.000,C 90.000,E1 95.391} C_DIS
LIN {X -0.134,Y -500.074,Z 1700.523,A 0.000,B 0.000,C 90.000,E1 94.188} C_DIS
LIN {X -0.003,Y -487.473,Z 1700.514,A 0.000,B 0.000,C 90.000,E1 92.465} C_DIS
LIN {X -0.141,Y -474.772,Z 1700.504,A 0.000,B 0.000,C 90.000,E1 90.745} C_DIS
LIN {X -0.069,Y -462.096,Z 1700.494,A 0.000,B 0.000,C 90.000,E1 88.969} C_DIS
LIN {X 0.212,Y -449.151,Z 1700.484,A 0.000,B 0.000,C 90.000,E1 87.135} C_DIS
LIN {X -0.197,Y -436.082,Z 1700.474,A 0.000,B 0.000,C 90.000,E1 85.355} C_DIS
LIN {X 0.088,Y -422.923,Z 1700.464,A 0.000,B 0.000,C 90.000,E1 83.451} C_DIS
LIN {X 0.219,Y -408.320,Z 1700.452,A 0.000,B 0.000,C 90.000,E1 81.254} C_DIS
LIN {X -0.123,Y -389.296,Z 1700.434,A 0.000,B 0.000,C 90.000,E1 78.229} C_DIS
LIN {X -0.105,Y -376.123,Z 1700.422,A 0.000,B 0.000,C 90.000,E1 75.936} C_DIS
LIN {X 0.140,Y -363.312,Z 1700.409,A 0.000,B 0.000,C 90.000,E1 73.559} C_DIS
LIN {X -0.128,Y -349.306,Z 1700.394,A 0.000,B 0.000,C 90.000,E1 70.913} C_DIS
LIN {X -0.098,Y -334.599,Z 1700.377,A 0.000,B 0.000,C 90.000,E1 67.847} C_DIS
LIN {X -0.080,Y -321.877,Z 1700.361,A 0.000,B 0.000,C 90.000,E1 65.025} C_DIS
LIN {X -0.192,Y -310.896,Z 1700.347,A 0.000,B 0.000,C 90.000,E1 62.487} C_DIS
LIN {X -0.174,Y -301.464,Z 1700.334,A 0.000,B 0.000,C 90.000,E1 60.205} C_DIS
LIN {X -0.069,Y -291.997,Z 1700.321,A 0.000,B 0.000,C 90.000,E1 57.867} C_DIS
LIN {X 0.163,Y -283.802,Z 1700.310,A 0.000,B 0.000,C 90.000,E1 55.801} C_DIS
LIN {X 0.004,Y -275.381,Z 1700.299,A 0.000,B 0.000,C 90.000,E1 53.783} C_DIS
LIN {X -0.047,Y -264.011,Z 1700.283,A 0.000,B 0.000,C 90.000,E1 51.009} C_DIS
LIN {X -0.072,Y -254.244,Z 1700.270,A 0.000,B 0.000,C 90.000,E1 48.528} C_DIS
LIN {X 0.003,Y -242.210,Z 1700.251,A 0.000,B 0.000,C 90.000,E1 45.243} C_DIS
LIN {X -0.048,Y -232.379,Z 1700.235,A 0.000,B 0.000,C 90.000,E1 42.285} C_DIS
LIN {X -0.070,Y -224.377,Z 1700.220,A 0.000,B 0.000,C 90.000,E1 39.644} C_DIS
LIN {X -0.117,Y -216.094,Z 1700.203,A 0.000,B 0.000,C 90.000,E1 36.583} C_DIS
LIN {X 0.024,Y -208.482,Z 1700.186,A 0.000,B 0.000,C 90.000,E1 33.420} C_DIS
LIN {X -0.023,Y -201.635,Z 1700.168,A 0.000,B 0.000,C 90.000,E1 30.256} C_DIS
LIN {X 0.085,Y -195.385,Z 1700.150,A 0.000,B 0.000,C 90.000,E1 27.001} C_DIS
LIN {X -0.044,Y -189.732,Z 1700.132,A 0.000,B 0.000,C 90.000,E1 23.770} C_DIS
LIN {X 0.062,Y -184.623,Z 1700.114,A 0.000,B 0.000,C 90.000,E1 20.429} C_DIS
LIN {X 0.019,Y -180.253,Z 1700.095,A 0.000,B 0.000,C 90.000,E1 17.094} C_DIS
LIN {X 0.010,Y -176.530,Z 1700.076,A 0.000,B 0.000,C 90.000,E1 13.716} C_DIS
LIN {X 0.034,Y -172.903,Z 1700.052,A 0.000,B 0.000,C 90.000,E1 9.443} C_DIS
LIN {X -0.031,Y -169.693,Z 1700.024,A 0.000,B 0.000,C 90.000,E1 4.302} C_DIS
LIN {X 0.056,Y -167.638,Z 1699.983,A 0.000,B 0.000,C 90.000,E1 356.906} C_DIS
LIN {X 0.088,Y -169.093,Z 1699.925,A 0.000,B 0.000,C 90.000,E1 346.464} C_DIS
LIN {X 0.082,Y -171.742,Z 1699.896,A 0.000,B 0.000,C 90.000,E1 341.275} C_DIS
LIN {X 0.020,Y -175.189,Z 1699.872,A 0.000,B 0.000,C 90.000,E1 336.997} C_DIS
LIN {X -0.006,Y -179.690,Z 1699.849,A 0.000,B 0.000,C 90.000,E1 332.743} C_DIS
LIN {X 0.106,Y -184.172,Z 1699.830,A 0.000,B 0.000,C 90.000,E1 329.331} C_DIS
LIN {X 0.065,Y -188.192,Z 1699.816,A 0.000,B 0.000,C 90.000,E1 326.834} C_DIS
LIN {X 0.038,Y -192.868,Z 1699.802,A 0.000,B 0.000,C 90.000,E1 324.356} C_DIS
LIN {X 0.007,Y -198.145,Z 1699.788,A 0.000,B 0.000,C 90.000,E1 321.904} C_DIS
LIN {X -0.071,Y -205.172,Z 1699.773,A 0.000,B 0.000,C 90.000,E1 319.094} C_DIS
LIN {X -0.025,Y -213.179,Z 1699.757,A 0.000,B 0.000,C 90.000,E1 316.296} C_DIS
LIN {X -0.018,Y -220.963,Z 1699.744,A 0.000,B 0.000,C 90.000,E1 313.947} C_DIS
LIN {X 0.096,Y -231.060,Z 1699.729,A 0.000,B 0.000,C 90.000,E1 311.229} C_DIS
LIN {X 0.033,Y -239.090,Z 1699.719,A 0.000,B 0.000,C 90.000,E1 309.358} C_DIS
LIN {X -0.051,Y -248.012,Z 1699.708,A 0.000,B 0.000,C 90.000,E1 307.523} C_DIS
LIN {X 0.081,Y -259.859,Z 1699.696,A 0.000,B 0.000,C 90.000,E1 305.311} C_DIS
LIN {X 0.006,Y -277.457,Z 1699.681,A 0.000,B 0.000,C 90.000,E1 302.498} C_DIS
LIN {X 0.097,Y -296.539,Z 1699.665,A 0.000,B 0.000,C 90.000,E1 299.745} C_DIS
LIN {X -0.079,Y -314.082,Z 1699.652,A 0.000,B 0.000,C 90.000,E1 297.462} C_DIS
LIN {X -0.111,Y -329.245,Z 1699.642,A 0.000,B 0.000,C 90.000,E1 295.540} C_DIS
LIN {X 0.002,Y -344.609,Z 1699.631,A 0.000,B 0.000,C 90.000,E1 293.643} C_DIS
LIN {X 0.101,Y -357.413,Z 1699.623,A 0.000,B 0.000,C 90.000,E1 292.099} C_DIS
LIN {X -0.011,Y -367.395,Z 1699.616,A 0.000,B 0.000,C 90.000,E1 290.918} C_DIS
LIN {X -0.141,Y -376.770,Z 1699.610,A 0.000,B 0.000,C 90.000,E1 289.758} C_DIS
LIN {X 0.071,Y -383.136,Z 1699.605,A 0.000,B 0.000,C 90.000,E1 288.852} C_DIS
LIN {X -0.011,Y -388.729,Z 1699.600,A 0.000,B 0.000,C 90.000,E1 288.000} C_DIS
LIN {X 0.168,Y -391.927,Z 1699.597,A 0.000,B 0.000,C 90.000,E1 287.402} C_DIS
LIN {X -0.006,Y -394.700,Z 1699.594,A 0.000,B 0.000,C 90.000,E1 286.858} C_DIS
LIN {X -0.108,Y -398.083,Z 1699.589,A 0.000,B 0.000,C 90.000,E1 286.024} C_DIS
LIN {X 0.137,Y -399.875,Z 1699.586,A 0.000,B 0.000,C 90.000,E1 285.426} C_DIS
LIN {X -0.104,Y -401.316,Z 1699.583,A 0.000,B 0.000,C 90.000,E1 284.898} C_DIS
LIN {X 0.157,Y -402.356,Z 1699.580,A 0.000,B 0.000,C 90.000,E1 284.300} C_DIS
LIN {X -0.062,Y -403.010,Z 1699.576,A 0.000,B 0.000,C 90.000,E1 283.772} C_DIS
LIN {X 0.210,Y -403.279,Z 1699.573,A 0.000,B 0.000,C 90.000,E1 283.175} C_DIS
LIN {X -0.001,Y -403.083,Z 1699.570,A 0.000,B 0.000,C 90.000,E1 282.647} C_DIS
LIN {X 0.185,Y -402.433,Z 1699.567,A 0.000,B 0.000,C 90.000,E1 282.063} C_DIS
LIN {X -0.025,Y -401.367,Z 1699.564,A 0.000,B 0.000,C 90.000,E1 281.535} C_DIS
LIN {X 0.155,Y -399.752,Z 1699.561,A 0.000,B 0.000,C 90.000,E1 280.950} C_DIS
LIN {X -0.066,Y -397.614,Z 1699.558,A 0.000,B 0.000,C 90.000,E1 280.423} C_DIS
LIN {X 0.027,Y -394.948,Z 1699.555,A 0.000,B 0.000,C 90.000,E1 279.849} C_DIS
LIN {X -0.160,Y -390.205,Z 1699.550,A 0.000,B 0.000,C 90.000,E1 279.029} C_DIS
LIN {X -0.023,Y -383.055,Z 1699.544,A 0.000,B 0.000,C 90.000,E1 277.871} C_DIS
LIN {X 0.011,Y -377.045,Z 1699.539,A 0.000,B 0.000,C 90.000,E1 277.004} C_DIS
LIN {X -0.011,Y -372.387,Z 1699.536,A 0.000,B 0.000,C 90.000,E1 276.429} C_DIS
LIN {X -0.059,Y -367.068,Z 1699.532,A 0.000,B 0.000,C 90.000,E1 275.853} C_DIS
LIN {X 0.024,Y -361.337,Z 1699.529,A 0.000,B 0.000,C 90.000,E1 275.277} C_DIS
LIN {X 0.014,Y -355.263,Z 1699.526,A 0.000,B 0.000,C 90.000,E1 274.759} C_DIS
LIN {X -0.077,Y -349.015,Z 1699.524,A 0.000,B 0.000,C 90.000,E1 274.302} C_DIS
LIN {X 0.148,Y -342.691,Z 1699.521,A 0.000,B 0.000,C 90.000,E1 273.841} C_DIS
LIN {X -0.086,Y -336.289,Z 1699.519,A 0.000,B 0.000,C 90.000,E1 273.498} C_DIS
LIN {X -0.006,Y -326.597,Z 1699.517,A 0.000,B 0.000,C 90.000,E1 272.980} C_DIS
LIN {X 0.098,Y -316.601,Z 1699.514,A 0.000,B 0.000,C 90.000,E1 272.522} C_DIS
LIN {X -0.073,Y -306.306,Z 1699.512,A 0.000,B 0.000,C 90.000,E1 272.178} C_DIS
LIN {X 0.069,Y -295.935,Z 1699.510,A 0.000,B 0.000,C 90.000,E1 271.835} C_DIS
LIN {X -0.120,Y -285.091,Z 1699.509,A 0.000,B 0.000,C 90.000,E1 271.604} C_DIS
LIN {X -0.070,Y -272.765,Z 1699.508,A 0.000,B 0.000,C 90.000,E1 271.375} C_DIS
LIN {X -0.094,Y -263.173,Z 1699.507,A 0.000,B 0.000,C 90.000,E1 271.260} C_DIS
LIN {X 0.119,Y -250.489,Z 1699.506,A 0.000,B 0.000,C 90.000,E1 271.146} C_DIS
LIN {X 0.063,Y -181.420,Z 1699.506,A 0.000,B 0.000,C 90.000,E1 271.146} C_DIS
LIN {X 0.026,Y -181.580,Z 1699.502,A 0.000,B 0.000,C 90.000,E1 270.286} C_DIS
LIN {X 0.002,Y -180.899,Z 1699.474,A 0.000,B 0.000,C 90.000,E1 265.241} C_DIS
LIN {X -0.049,Y -180.218,Z 1699.464,A 0.000,B 0.000,C 90.000,E1 263.571} C_DIS
LIN {X 0.081,Y -179.035,Z 1699.445,A 0.000,B 0.000,C 90.000,E1 260.151} C_DIS
LIN {X -0.032,Y -178.696,Z 1699.441,A 0.000,B 0.000,C 90.000,E1 259.342} C_DIS
LIN {X 0.078,Y -175.745,Z 1699.412,A 0.000,B 0.000,C 90.000,E1 254.212} C_DIS
LIN {X 0.073,Y -171.928,Z 1699.384,A 0.000,B 0.000,C 90.000,E1 249.082} C_DIS
LIN {X 0.048,Y -171.304,Z 1699.379,A 0.000,B 0.000,C 90.000,E1 248.230} C_DIS
LIN {X 0.093,Y -167.565,Z 1699.355,A 0.000,B 0.000,C 90.000,E1 243.896} C_DIS
LIN {X 0.106,Y -166.193,Z 1699.345,A 0.000,B 0.000,C 90.000,E1 242.153} C_DIS
LIN {X 0.096,Y -162.961,Z 1699.326,A 0.000,B 0.000,C 90.000,E1 238.663} C_DIS
LIN {X -0.081,Y -160.871,Z 1699.311,A 0.000,B 0.000,C 90.000,E1 236.087} C_DIS
LIN {X -0.102,Y -157.644,Z 1699.292,A 0.000,B 0.000,C 90.000,E1 232.557} C_DIS
LIN {X 0.057,Y -155.681,Z 1699.277,A 0.000,B 0.000,C 90.000,E1 229.828} C_DIS
LIN {X 0.001,Y -151.948,Z 1699.252,A 0.000,B 0.000,C 90.000,E1 225.364} C_DIS
LIN {X -0.090,Y -150.186,Z 1699.237,A 0.000,B 0.000,C 90.000,E1 222.690} C_DIS
LIN {X 0.042,Y -146.959,Z 1699.212,A 0.000,B 0.000,C 90.000,E1 218.096} C_DIS
LIN {X -0.055,Y -145.546,Z 1699.197,A 0.000,B 0.000,C 90.000,E1 215.391} C_DIS
LIN {X -0.055,Y -142.941,Z 1699.171,A 0.000,B 0.000,C 90.000,E1 210.797} C_DIS
LIN {X 0.003,Y -141.565,Z 1699.150,A 0.000,B 0.000,C 90.000,E1 207.078} C_DIS
LIN {X 0.055,Y -139.411,Z 1699.114,A 0.000,B 0.000,C 90.000,E1 200.556} C_DIS
LIN {X -0.023,Y -139.133,Z 1699.104,A 0.000,B 0.000,C 90.000,E1 198.725} C_DIS
LIN {X 0.004,Y -138.350,Z 1699.057,A 0.000,B 0.000,C 90.000,E1 190.310} C_DIS
LIN {X -0.008,Y -139.496,Z 1699.005,A 0.000,B 0.000,C 90.000,E1 180.974} C_DIS
LIN {X -0.068,Y -141.116,Z 1698.974,A 0.000,B 0.000,C 90.000,E1 175.412} C_DIS
LIN {X 0.026,Y -142.495,Z 1698.959,A 0.000,B 0.000,C 90.000,E1 172.591} C_DIS
LIN {X -0.027,Y -144.748,Z 1698.933,A 0.000,B 0.000,C 90.000,E1 167.993} C_DIS
LIN {X -0.078,Y -147.357,Z 1698.913,A 0.000,B 0.000,C 90.000,E1 164.338} C_DIS
LIN {X -0.013,Y -150.683,Z 1698.887,A 0.000,B 0.000,C 90.000,E1 159.752} C_DIS
LIN {X 0.070,Y -154.163,Z 1698.867,A 0.000,B 0.000,C 90.000,E1 156.102} C_DIS
LIN {X 0.000,Y -157.595,Z 1698.847,A 0.000,B 0.000,C 90.000,E1 152.538} C_DIS
LIN {X -0.049,Y -161.846,Z 1698.828,A 0.000,B 0.000,C 90.000,E1 148.997} C_DIS
LIN {X -0.031,Y -166.037,Z 1698.808,A 0.000,B 0.000,C 90.000,E1 145.468} C_DIS
LIN {X -0.040,Y -171.039,Z 1698.789,A 0.000,B 0.000,C 90.000,E1 141.984} C_DIS
LIN {X -0.009,Y -175.910,Z 1698.770,A 0.000,B 0.000,C 90.000,E1 138.528} C_DIS
LIN {X -0.017,Y -180.147,Z 1698.755,A 0.000,B 0.000,C 90.000,E1 135.972} C_DIS
LIN {X -0.047,Y -185.565,Z 1698.737,A 0.000,B 0.000,C 90.000,E1 132.609} C_DIS
LIN {X 0.003,Y -190.153,Z 1698.723,A 0.000,B 0.000,C 90.000,E1 130.092} C_DIS
LIN {X 0.021,Y -195.923,Z 1698.704,A 0.000,B 0.000,C 90.000,E1 126.790} C_DIS
LIN {X 0.090,Y -200.753,Z 1698.691,A 0.000,B 0.000,C 90.000,E1 124.326} C_DIS
LIN {X 0.002,Y -206.642,Z 1698.673,A 0.000,B 0.000,C 90.000,E1 121.131} C_DIS
LIN {X -0.049,Y -208.818,Z 1698.667,A 0.000,B 0.000,C 90.000,E1 120.079} C_DIS
LIN {X 0.044,Y -331.174,Z 1698.667,A 0.000,B 0.000,C 90.000,E1 120.050} C_DIS
LIN {X -0.045,Y -332.920,Z 1698.667,A 0.000,B 0.000,C 90.000,E1 120.050} C_DIS
LIN {X -0.029,Y -338.853,Z 1698.666,A 0.000,B 0.000,C 90.000,E1 119.795} C_DIS
LIN {X -0.011,Y -341.760,Z 1698.664,A 0.000,B 0.000,C 90.000,E1 119.539} C_DIS
LIN {X 0.096,Y -345.447,Z 1698.661,A 0.000,B 0.000,C 90.000,E1 119.027} C_DIS
LIN {X -0.057,Y -348.397,Z 1698.658,A 0.000,B 0.000,C 90.000,E1 118.437} C_DIS
LIN {X -0.093,Y -361.253,Z 1698.643,A 0.000,B 0.000,C 90.000,E1 115.720} C_DIS
LIN {X 0.095,Y -375.634,Z 1698.628,A 0.000,B 0.000,C 90.000,E1 113.025} C_DIS
LIN {X -0.092,Y -389.791,Z 1698.615,A 0.000,B 0.000,C 90.000,E1 110.737} C_DIS
LIN {X -0.084,Y -405.343,Z 1698.603,A 0.000,B 0.000,C 90.000,E1 108.471} C_DIS
LIN {X -0.082,Y -422.398,Z 1698.590,A 0.000,B 0.000,C 90.000,E1 106.260} C_DIS
LIN {X -0.184,Y -441.074,Z 1698.578,A 0.000,B 0.000,C 90.000,E1 104.120} C_DIS
LIN {X -0.076,Y -460.960,Z 1698.567,A 0.000,B 0.000,C 90.000,E1 102.063} C_DIS
LIN {X -0.070,Y -483.981,Z 1698.555,A 0.000,B 0.000,C 90.000,E1 99.962} C_DIS
LIN {X 0.209,Y -504.877,Z 1698.546,A 0.000,B 0.000,C 90.000,E1 98.219} C_DIS
LIN {X -0.100,Y -506.855,Z 1698.545,A 0.000,B 0.000,C 90.000,E1 98.049} C_DIS
LIN {X -0.160,Y -508.619,Z 1698.543,A 0.000,B 0.000,C 90.000,E1 97.814} C_DIS
LIN {X 0.217,Y -509.937,Z 1698.542,A 0.000,B 0.000,C 90.000,E1 97.530} C_DIS
LIN {X 0.051,Y -511.561,Z 1698.539,A 0.000,B 0.000,C 90.000,E1 97.068} C_DIS
LIN {X -0.108,Y -512.085,Z 1698.537,A 0.000,B 0.000,C 90.000,E1 96.606} C_DIS
LIN {X -0.257,Y -511.593,Z 1698.534,A 0.000,B 0.000,C 90.000,E1 96.144} C_DIS
LIN {X 0.103,Y -510.004,Z 1698.531,A 0.000,B 0.000,C 90.000,E1 95.625} C_DIS
LIN {X 0.051,Y -508.707,Z 1698.530,A 0.000,B 0.000,C 90.000,E1 95.391} C_DIS
LIN {X 0.058,Y -499.922,Z 1698.523,A 0.000,B 0.000,C 90.000,E1 94.188} C_DIS
LIN {X 0.181,Y -487.332,Z 1698.514,A 0.000,B 0.000,C 90.000,E1 92.465} C_DIS
LIN {X 0.036,Y -474.637,Z 1698.504,A 0.000,B 0.000,C 90.000,E1 90.745} C_DIS
LIN {X 0.100,Y -461.966,Z 1698.494,A 0.000,B 0.000,C 90.000,E1 88.969} C_DIS
LIN {X -0.075,Y -449.041,Z 1698.484,A 0.000,B 0.000,C 90.000,E1 87.192} C_DIS
LIN {X -0.042,Y -435.954,Z 1698.474,A 0.000,B 0.000,C 90.000,E1 85.355} C_DIS
LIN {X 0.187,Y -422.751,Z 1698.464,A 0.000,B 0.000,C 90.000,E1 83.457} C_DIS
LIN {X -0.107,Y -408.128,Z 1698.452,A 0.000,B 0.000,C 90.000,E1 81.319} C_DIS
LIN {X 0.003,Y -389.082,Z 1698.435,A 0.000,B 0.000,C 90.000,E1 78.229} C_DIS
LIN {X 0.011,Y -375.879,Z 1698.422,A 0.000,B 0.000,C 90.000,E1 75.936} C_DIS
LIN {X -0.102,Y -363.043,Z 1698.409,A 0.000,B 0.000,C 90.000,E1 73.614} C_DIS
LIN {X -0.034,Y -349.020,Z 1698.394,A 0.000,B 0.000,C 90.000,E1 70.913} C_DIS
LIN {X -0.016,Y -334.305,Z 1698.377,A 0.000,B 0.000,C 90.000,E1 67.847} C_DIS
LIN {X -0.010,Y -321.616,Z 1698.361,A 0.000,B 0.000,C 90.000,E1 65.025} C_DIS
LIN {X -0.129,Y -310.636,Z 1698.347,A 0.000,B 0.000,C 90.000,E1 62.487} C_DIS
LIN {X -0.118,Y -301.220,Z 1698.334,A 0.000,B 0.000,C 90.000,E1 60.205} C_DIS
LIN {X -0.019,Y -293.113,Z 1698.323,A 0.000,B 0.000,C 90.000,E1 58.201} C_DIS
LIN {X 0.075,Y -284.934,Z 1698.312,A 0.000,B 0.000,C 90.000,E1 56.167} C_DIS
LIN {X 0.097,Y -276.503,Z 1698.301,A 0.000,B 0.000,C 90.000,E1 54.116} C_DIS
LIN {X 0.042,Y -266.534,Z 1698.287,A 0.000,B 0.000,C 90.000,E1 51.698} C_DIS
LIN {X 0.101,Y -255.346,Z 1698.271,A 0.000,B 0.000,C 90.000,E1 48.852} C_DIS
LIN {X -0.145,Y -243.228,Z 1698.253,A 0.000,B 0.000,C 90.000,E1 45.648} C_DIS
LIN {X -0.005,Y -233.312,Z 1698.237,A 0.000,B 0.000,C 90.000,E1 42.651} C_DIS
LIN {X -0.070,Y -224.179,Z 1698.220,A 0.000,B 0.000,C 90.000,E1 39.644} C_DIS
LIN {X -0.122,Y -215.926,Z 1698.203,A 0.000,B 0.000,C 90.000,E1 36.583} C_DIS
LIN {X 0.015,Y -208.364,Z 1698.186,A 0.000,B 0.000,C 90.000,E1 33.420} C_DIS
LIN {X -0.035,Y -201.531,Z 1698.168,A 0.000,B 0.000,C 90.000,E1 30.256} C_DIS
LIN {X 0.072,Y -195.303,Z 1698.150,A 0.000,B 0.000,C 90.000,E1 27.001} C_DIS
LIN {X -0.058,Y -189.656,Z 1698.132,A 0.000,B 0.000,C 90.000,E1 23.770} C_DIS
LIN {X 0.045,Y -184.579,Z 1698.114,A 0.000,B 0.000,C 90.000,E1 20.429} C_DIS
LIN {X 0.002,Y -180.204,Z 1698.095,A 0.000,B 0.000,C 90.000,E1 17.094} C_DIS
LIN {X -0.008,Y -176.485,Z 1698.076,A 0.000,B 0.000,C 90.000,E1 13.716} C_DIS
LIN {X 0.015,Y -172.863,Z 1698.052,A 0.000,B 0.000,C 90.000,E1 9.443} C_DIS
LIN {X -0.051,Y -169.648,Z 1698.024,A 0.000,B 0.000,C 90.000,E1 4.302} C_DIS
LIN {X 0.055,Y -167.562,Z 1697.983,A 0.000,B 0.000,C 90.000,E1 356.906} C_DIS
LIN {X 0.082,Y -169.022,Z 1697.925,A 0.000,B 0.000,C 90.000,E1 346.464} C_DIS
LIN {X 0.073,Y -171.685,Z 1697.896,A 0.000,B 0.000,C 90.000,E1 341.275} C_DIS
LIN {X 0.009,Y -175.148,Z 1697.872,A 0.000,B 0.000,C 90.000,E1 336.997} C_DIS
LIN {X -0.019,Y -179.711,Z 1697.849,A 0.000,B 0.000,C 90.000,E1 332.743} C_DIS
LIN {X 0.095,Y -184.230,Z 1697.830,A 0.000,B 0.000,C 90.000,E1 329.331} C_DIS
LIN {X 0.054,Y -188.272,Z 1697.816,A 0.000,B 0.000,C 90.000,E1 326.834} C_DIS
LIN {X -0.006,Y -194.669,Z 1697.797,A 0.000,B 0.000,C 90.000,E1 323.543} C_DIS
LIN {X 0.022,Y -201.199,Z 1697.782,A 0.000,B 0.000,C 90.000,E1 320.678} C_DIS
LIN {X -0.009,Y -208.640,Z 1697.766,A 0.000,B 0.000,C 90.000,E1 317.877} C_DIS
LIN {X 0.117,Y -217.130,Z 1697.751,A 0.000,B 0.000,C 90.000,E1 315.081} C_DIS
LIN {X -0.021,Y -226.805,Z 1697.736,A 0.000,B 0.000,C 90.000,E1 312.405} C_DIS
LIN {X 0.114,Y -235.980,Z 1697.723,A 0.000,B 0.000,C 90.000,E1 310.092} C_DIS
LIN {X -0.033,Y -246.381,Z 1697.710,A 0.000,B 0.000,C 90.000,E1 307.890} C_DIS
LIN {X 0.068,Y -258.020,Z 1697.698,A 0.000,B 0.000,C 90.000,E1 305.678} C_DIS
LIN {X 0.098,Y -275.328,Z 1697.682,A 0.000,B 0.000,C 90.000,E1 302.832} C_DIS
LIN {X -0.117,Y -294.228,Z 1697.667,A 0.000,B 0.000,C 90.000,E1 300.129} C_DIS
LIN {X 0.067,Y -311.657,Z 1697.654,A 0.000,B 0.000,C 90.000,E1 297.769} C_DIS
LIN {X -0.011,Y -326.774,Z 1697.644,A 0.000,B 0.000,C 90.000,E1 295.848} C_DIS
LIN {X 0.125,Y -341.986,Z 1697.633,A 0.000,B 0.000,C 90.000,E1 293.951} C_DIS
LIN {X -0.115,Y -357.350,Z 1697.623,A 0.000,B 0.000,C 90.000,E1 292.153} C_DIS
LIN {X 0.107,Y -367.321,Z 1697.616,A 0.000,B 0.000,C 90.000,E1 290.918} C_DIS
LIN {X -0.021,Y -376.700,Z 1697.610,A 0.000,B 0.000,C 90.000,E1 289.758} C_DIS
LIN {X -0.170,Y -383.130,Z 1697.605,A 0.000,B 0.000,C 90.000,E1 288.906} C_DIS
LIN {X 0.112,Y -388.746,Z 1697.600,A 0.000,B 0.000,C 90.000,E1 288.000} C_DIS
LIN {X -0.045,Y -393.368,Z 1697.595,A 0.000,B 0.000,C 90.000,E1 287.166} C_DIS
LIN {X -0.211,Y -395.953,Z 1697.592,A 0.000,B 0.000,C 90.000,E1 286.622} C_DIS
LIN {X 0.019,Y -398.132,Z 1697.589,A 0.000,B 0.000,C 90.000,E1 286.024} C_DIS
LIN {X -0.122,Y -399.962,Z 1697.586,A 0.000,B 0.000,C 90.000,E1 285.481} C_DIS
LIN {X 0.024,Y -401.433,Z 1697.583,A 0.000,B 0.000,C 90.000,E1 284.898} C_DIS
LIN {X -0.104,Y -402.498,Z 1697.580,A 0.000,B 0.000,C 90.000,E1 284.356} C_DIS
LIN {X 0.067,Y -403.162,Z 1697.577,A 0.000,B 0.000,C 90.000,E1 283.772} C_DIS
LIN {X -0.145,Y -403.448,Z 1697.573,A 0.000,B 0.000,C 90.000,E1 283.244} C_DIS
LIN {X 0.131,Y -403.306,Z 1697.570,A 0.000,B 0.000,C 90.000,E1 282.647} C_DIS
LIN {X -0.077,Y -402.723,Z 1697.567,A 0.000,B 0.000,C 90.000,E1 282.119} C_DIS
LIN {X 0.109,Y -401.673,Z 1697.564,A 0.000,B 0.000,C 90.000,E1 281.535} C_DIS
LIN {X -0.103,Y -400.053,Z 1697.561,A 0.000,B 0.000,C 90.000,E1 281.007} C_DIS
LIN {X -0.002,Y -397.974,Z 1697.558,A 0.000,B 0.000,C 90.000,E1 280.433} C_DIS
LIN {X 0.163,Y -395.333,Z 1697.555,A 0.000,B 0.000,C 90.000,E1 279.849} C_DIS
LIN {X -0.022,Y -390.580,Z 1697.550,A 0.000,B 0.000,C 90.000,E1 279.029} C_DIS
LIN {X 0.116,Y -383.430,Z 1697.544,A 0.000,B 0.000,C 90.000,E1 277.871} C_DIS
LIN {X 0.106,Y -377.393,Z 1697.539,A 0.000,B 0.000,C 90.000,E1 277.011} C_DIS
LIN {X 0.129,Y -372.679,Z 1697.536,A 0.000,B 0.000,C 90.000,E1 276.429} C_DIS
LIN {X 0.082,Y -367.343,Z 1697.533,A 0.000,B 0.000,C 90.000,E1 275.853} C_DIS
LIN {X -0.159,Y -361.630,Z 1697.530,A 0.000,B 0.000,C 90.000,E1 275.334} C_DIS
LIN {X -0.139,Y -355.626,Z 1697.527,A 0.000,B 0.000,C 90.000,E1 274.816} C_DIS
LIN {X 0.118,Y -349.344,Z 1697.524,A 0.000,B 0.000,C 90.000,E1 274.302} C_DIS
LIN {X -0.097,Y -339.893,Z 1697.521,A 0.000,B 0.000,C 90.000,E1 273.726} C_DIS
LIN {X 0.120,Y -330.029,Z 1697.518,A 0.000,B 0.000,C 90.000,E1 273.154} C_DIS
LIN {X 0.152,Y -320.306,Z 1697.515,A 0.000,B 0.000,C 90.000,E1 272.694} C_DIS
LIN {X 0.128,Y -310.000,Z 1697.513,A 0.000,B 0.000,C 90.000,E1 272.293} C_DIS
LIN {X -0.112,Y -299.735,Z 1697.511,A 0.000,B 0.000,C 90.000,E1 272.007} C_DIS
LIN {X -0.122,Y -289.149,Z 1697.509,A 0.000,B 0.000,C 90.000,E1 271.718} C_DIS
LIN {X -0.070,Y -281.599,Z 1697.509,A 0.000,B 0.000,C 90.000,E1 271.547} C_DIS
LIN {X 0.068,Y -268.868,Z 1697.507,A 0.000,B 0.000,C 90.000,E1 271.318} C_DIS
LIN {X 0.104,Y -257.312,Z 1697.507,A 0.000,B 0.000,C 90.000,E1 271.203} C_DIS
LIN {X 0.005,Y -251.128,Z 1697.507,A 0.000,B 0.000,C 90.000,E1 271.203} C_DIS
LIN {X -0.019,Y -186.571,Z 1697.507,A 0.000,B 0.000,C 90.000,E1 271.203} C_DIS
LIN {X -0.042,Y -181.751,Z 1697.507,A 0.000,B 0.000,C 90.000,E1 271.203} C_DIS
LIN {X -0.065,Y -181.416,Z 1697.507,A 0.000,B 0.000,C 90.000,E1 271.203} C_DIS
LIN {X -0.037,Y -181.578,Z 1697.501,A 0.000,B 0.000,C 90.000,E1 270.172} C_DIS
LIN {X -0.034,Y -180.848,Z 1697.472,A 0.000,B 0.000,C 90.000,E1 264.951} C_DIS
LIN {X 0.049,Y -178.957,Z 1697.444,A 0.000,B 0.000,C 90.000,E1 259.859} C_DIS
LIN {X -0.059,Y -177.359,Z 1697.430,A 0.000,B 0.000,C 90.000,E1 257.353} C_DIS
LIN {X 0.036,Y -175.531,Z 1697.411,A 0.000,B 0.000,C 90.000,E1 253.921} C_DIS
LIN {X 0.038,Y -172.266,Z 1697.387,A 0.000,B 0.000,C 90.000,E1 249.645} C_DIS
LIN {X 0.077,Y -171.745,Z 1697.382,A 0.000,B 0.000,C 90.000,E1 248.773} C_DIS
LIN {X -0.065,Y -167.343,Z 1697.353,A 0.000,B 0.000,C 90.000,E1 243.640} C_DIS
LIN {X 0.017,Y -166.730,Z 1697.349,A 0.000,B 0.000,C 90.000,E1 242.743} C_DIS
LIN {X -0.070,Y -162.709,Z 1697.324,A 0.000,B 0.000,C 90.000,E1 238.408} C_DIS
LIN {X -0.009,Y -161.399,Z 1697.315,A 0.000,B 0.000,C 90.000,E1 236.628} C_DIS
LIN {X 0.033,Y -157.393,Z 1697.290,A 0.000,B 0.000,C 90.000,E1 232.190} C_DIS
LIN {X -0.034,Y -155.389,Z 1697.275,A 0.000,B 0.000,C 90.000,E1 229.542} C_DIS
LIN {X 0.006,Y -151.724,Z 1697.250,A 0.000,B 0.000,C 90.000,E1 225.040} C_DIS
LIN {X 0.021,Y -149.919,Z 1697.235,A 0.000,B 0.000,C 90.000,E1 222.324} C_DIS
LIN {X -0.060,Y -146.771,Z 1697.210,A 0.000,B 0.000,C 90.000,E1 217.810} C_DIS
LIN {X 0.043,Y -145.342,Z 1697.195,A 0.000,B 0.000,C 90.000,E1 215.025} C_DIS
LIN {X -0.041,Y -142.418,Z 1697.164,A 0.000,B 0.000,C 90.000,E1 209.539} C_DIS
LIN {X 0.008,Y -141.405,Z 1697.149,A 0.000,B 0.000,C 90.000,E1 206.744} C_DIS
LIN {X -0.004,Y -139.357,Z 1697.112,A 0.000,B 0.000,C 90.000,E1 200.248} C_DIS
LIN {X -0.017,Y -138.797,Z 1697.097,A 0.000,B 0.000,C 90.000,E1 197.457} C_DIS
LIN {X 0.038,Y -138.348,Z 1697.055,A 0.000,B 0.000,C 90.000,E1 189.962} C_DIS
LIN {X 0.056,Y -139.372,Z 1697.009,A 0.000,B 0.000,C 90.000,E1 181.547} C_DIS
LIN {X -0.031,Y -141.261,Z 1696.973,A 0.000,B 0.000,C 90.000,E1 175.065} C_DIS
LIN {X 0.068,Y -142.628,Z 1696.957,A 0.000,B 0.000,C 90.000,E1 172.243} C_DIS
LIN {X 0.020,Y -144.953,Z 1696.931,A 0.000,B 0.000,C 90.000,E1 167.645} C_DIS
LIN {X 0.012,Y -147.581,Z 1696.911,A 0.000,B 0.000,C 90.000,E1 163.976} C_DIS
LIN {X 0.042,Y -150.193,Z 1696.891,A 0.000,B 0.000,C 90.000,E1 160.315} C_DIS
LIN {X -0.032,Y -153.574,Z 1696.871,A 0.000,B 0.000,C 90.000,E1 156.719} C_DIS
LIN {X -0.041,Y -156.991,Z 1696.851,A 0.000,B 0.000,C 90.000,E1 153.127} C_DIS
LIN {X 0.032,Y -161.105,Z 1696.831,A 0.000,B 0.000,C 90.000,E1 149.537} C_DIS
LIN {X -0.023,Y -163.208,Z 1696.821,A 0.000,B 0.000,C 90.000,E1 147.788} C_DIS
LIN {X -0.017,Y -167.636,Z 1696.802,A 0.000,B 0.000,C 90.000,E1 144.276} C_DIS
LIN {X -0.004,Y -171.461,Z 1696.787,A 0.000,B 0.000,C 90.000,E1 141.662} C_DIS
LIN {X -0.073,Y -176.388,Z 1696.768,A 0.000,B 0.000,C 90.000,E1 138.243} C_DIS
LIN {X 0.049,Y -180.680,Z 1696.754,A 0.000,B 0.000,C 90.000,E1 135.648} C_DIS
LIN {X 0.031,Y -186.083,Z 1696.735,A 0.000,B 0.000,C 90.000,E1 132.285} C_DIS
LIN {X -0.033,Y -190.720,Z 1696.721,A 0.000,B 0.000,C 90.000,E1 129.806} C_DIS
LIN {X -0.001,Y -196.473,Z 1696.703,A 0.000,B 0.000,C 90.000,E1 126.503} C_DIS
LIN {X -0.035,Y -201.253,Z 1696.689,A 0.000,B 0.000,C 90.000,E1 124.072} C_DIS
LIN {X -0.025,Y -207.585,Z 1696.670,A 0.000,B 0.000,C 90.000,E1 120.669} C_DIS
LIN {X 0.066,Y -208.751,Z 1696.667,A 0.000,B 0.000,C 90.000,E1 120.079} C_DIS
LIN {X 0.071,Y -331.530,Z 1696.667,A 0.000,B 0.000,C 90.000,E1 120.079} C_DIS
LIN {X -0.014,Y -334.110,Z 1696.667,A 0.000,B 0.000,C 90.000,E1 120.050} C_DIS
LIN {X -0.098,Y -337.433,Z 1696.666,A 0.000,B 0.000,C 90.000,E1 119.922} C_DIS
LIN {X -0.155,Y -340.910,Z 1696.665,A 0.000,B 0.000,C 90.000,E1 119.667} C_DIS
LIN {X -0.055,Y -344.543,Z 1696.662,A 0.000,B 0.000,C 90.000,E1 119.205} C_DIS
LIN {X 0.100,Y -346.305,Z 1696.661,A 0.000,B 0.000,C 90.000,E1 118.871} C_DIS
LIN {X 0.038,Y -360.481,Z 1696.644,A 0.000,B 0.000,C 90.000,E1 115.848} C_DIS
LIN {X -0.135,Y -374.775,Z 1696.629,A 0.000,B 0.000,C 90.000,E1 113.206} C_DIS
LIN {X 0.009,Y -388.848,Z 1696.616,A 0.000,B 0.000,C 90.000,E1 110.865} C_DIS
LIN {X 0.001,Y -404.311,Z 1696.603,A 0.000,B 0.000,C 90.000,E1 108.598} C_DIS
LIN {X -0.014,Y -421.269,Z 1696.591,A 0.000,B 0.000,C 90.000,E1 106.386} C_DIS
LIN {X -0.134,Y -439.840,Z 1696.579,A 0.000,B 0.000,C 90.000,E1 104.245} C_DIS
LIN {X -0.005,Y -459.690,Z 1696.568,A 0.000,B 0.000,C 90.000,E1 102.175} C_DIS
LIN {X -0.095,Y -482.675,Z 1696.556,A 0.000,B 0.000,C 90.000,E1 100.074} C_DIS
LIN {X 0.027,Y -503.636,Z 1696.546,A 0.000,B 0.000,C 90.000,E1 98.341} C_DIS
LIN {X -0.219,Y -505.874,Z 1696.545,A 0.000,B 0.000,C 90.000,E1 98.163} C_DIS
LIN {X -0.236,Y -507.739,Z 1696.544,A 0.000,B 0.000,C 90.000,E1 97.936} C_DIS
LIN {X -0.184,Y -509.153,Z 1696.543,A 0.000,B 0.000,C 90.000,E1 97.701} C_DIS
LIN {X 0.150,Y -511.062,Z 1696.540,A 0.000,B 0.000,C 90.000,E1 97.182} C_DIS
LIN {X -0.014,Y -511.823,Z 1696.537,A 0.000,B 0.000,C 90.000,E1 96.720} C_DIS
LIN {X -0.168,Y -511.564,Z 1696.535,A 0.000,B 0.000,C 90.000,E1 96.258} C_DIS
LIN {X 0.190,Y -510.244,Z 1696.532,A 0.000,B 0.000,C 90.000,E1 95.739} C_DIS
LIN {X 0.090,Y -509.117,Z 1696.531,A 0.000,B 0.000,C 90.000,E1 95.511} C_DIS
LIN {X 0.038,Y -507.595,Z 1696.529,A 0.000,B 0.000,C 90.000,E1 95.277} C_DIS
LIN {X -0.058,Y -496.943,Z 1696.521,A 0.000,B 0.000,C 90.000,E1 93.841} C_DIS
LIN {X 0.134,Y -486.162,Z 1696.513,A 0.000,B 0.000,C 90.000,E1 92.350} C_DIS
LIN {X -0.038,Y -473.457,Z 1696.503,A 0.000,B 0.000,C 90.000,E1 90.630} C_DIS
LIN {X 0.011,Y -460.785,Z 1696.494,A 0.000,B 0.000,C 90.000,E1 88.854} C_DIS
LIN {X -0.190,Y -447.857,Z 1696.484,A 0.000,B 0.000,C 90.000,E1 87.078} C_DIS
LIN {X -0.175,Y -434.731,Z 1696.473,A 0.000,B 0.000,C 90.000,E1 85.241} C_DIS
LIN {X 0.180,Y -419.670,Z 1696.462,A 0.000,B 0.000,C 90.000,E1 83.053} C_DIS
LIN {X -0.118,Y -405.115,Z 1696.449,A 0.000,B 0.000,C 90.000,E1 80.905} C_DIS
LIN {X -0.087,Y -386.235,Z 1696.432,A 0.000,B 0.000,C 90.000,E1 77.813} C_DIS
LIN {X -0.137,Y -373.072,Z 1696.419,A 0.000,B 0.000,C 90.000,E1 75.519} C_DIS
LIN {X 0.036,Y -360.287,Z 1696.406,A 0.000,B 0.000,C 90.000,E1 73.142} C_DIS
LIN {X 0.131,Y -346.348,Z 1696.391,A 0.000,B 0.000,C 90.000,E1 70.423} C_DIS
LIN {X 0.063,Y -331.786,Z 1696.374,A 0.000,B 0.000,C 90.000,E1 67.358} C_DIS
LIN {X -0.009,Y -319.199,Z 1696.359,A 0.000,B 0.000,C 90.000,E1 64.537} C_DIS
LIN {X -0.006,Y -306.911,Z 1696.342,A 0.000,B 0.000,C 90.000,E1 61.641} C_DIS
LIN {X 0.048,Y -298.882,Z 1696.332,A 0.000,B 0.000,C 90.000,E1 59.665} C_DIS
LIN {X 0.090,Y -289.350,Z 1696.319,A 0.000,B 0.000,C 90.000,E1 57.327} C_DIS
LIN {X 0.035,Y -281.086,Z 1696.307,A 0.000,B 0.000,C 90.000,E1 55.308} C_DIS
LIN {X -0.008,Y -272.528,Z 1696.296,A 0.000,B 0.000,C 90.000,E1 53.256} C_DIS
LIN {X 0.022,Y -262.604,Z 1696.282,A 0.000,B 0.000,C 90.000,E1 50.803} C_DIS
LIN {X -0.043,Y -252.872,Z 1696.268,A 0.000,B 0.000,C 90.000,E1 48.324} C_DIS
LIN {X -0.011,Y -240.949,Z 1696.250,A 0.000,B 0.000,C 90.000,E1 45.040} C_DIS
LIN {X -0.084,Y -231.230,Z 1696.234,A 0.000,B 0.000,C 90.000,E1 42.081} C_DIS
LIN {X -0.046,Y -222.299,Z 1696.217,A 0.000,B 0.000,C 90.000,E1 39.036} C_DIS
